LIN {X 0,Y 149.454,Z 1124.639,A -85,B 0,C 180,E1 26452.481,E2 26452.481} C_VEL
LIN {X 0,Y 187.503,Z 1102.336,A -85,B 0,C 180,E1 26457.86,E2 26457.86} C_VEL
LIN {X 0,Y 200.138,Z 1093.431,A -85,B 0,C 180,E1 26459.166,E2 26459.166} C_VEL
LIN {X 0,Y 164.642,Z 1117.097,A -85,B 0,C 180,E1 26463.123,E2 26463.123} C_VEL
LIN {X 0,Y 149.261,Z 1125.368,A -85,B 0,C 180,E1 26463.863,E2 26463.863} C_VEL
LIN {X 0,Y 133.576,Z 1132.787,A -85,B 0,C 180,E1 26464.835,E2 26464.835} C_VEL
LIN {X 0,Y 93.97,Z 1148.455,A -85,B 0,C 180,E1 26475.529,E2 26475.529} C_VEL
LIN {X 0,Y 59.436,Z 1158.376,A -85,B 0,C 180,E1 26500.391,E2 26500.391} C_VEL
LIN {X 0,Y 47.074,Z 1161.431,A -85,B 0,C 180,E1 26534.085,E2 26534.085} C_VEL
LIN {X 0,Y 46.801,Z 1161.776,A -85,B 0,C 180,E1 26550.002,E2 26550.002} C_VEL
LIN {X 0,Y 51.769,Z 1160.244,A -85,B 0,C 180,E1 26585.663,E2 26585.663} C_VEL
LIN {X 0,Y 74.671,Z 1154.337,A -85,B 0,C 180,E1 26614.388,E2 26614.388} C_VEL
LIN {X 0,Y 111.047,Z 1142.33,A -85,B 0,C 180,E1 26630.135,E2 26630.135} C_VEL
LIN {X 0,Y 148.291,Z 1125.731,A -85,B 0,C 180,E1 26637.593,E2 26637.593} C_VEL
LIN {X 0,Y 174.697,Z 1110.81,A -85,B 0,C 180,E1 26640.902,E2 26640.902} C_VEL
LIN {X 0,Y 136.275,Z 1130.859,A -85,B 0,C 180,E1 26646.357,E2 26646.357} C_VEL
LIN {X 0,Y 98.213,Z 1145.413,A -85,B 0,C 180,E1 26656.197,E2 26656.197} C_VEL
LIN {X 0,Y 70.679,Z 1153.183,A -85,B 0,C 180,E1 26671.347,E2 26671.347} C_VEL
LIN {X 0,Y 52.791,Z 1157.045,A -85,B 0,C 180,E1 26695.129,E2 26695.129} C_VEL
LIN {X 0,Y 47.067,Z 1158.256,A -85,B 0,C 180,E1 26729.998,E2 26729.998} C_VEL
LIN {X 0,Y 52.803,Z 1157.02,A -85,B 0,C 180,E1 26764.857,E2 26764.857} C_VEL
LIN {X 0,Y 76.325,Z 1151.652,A -85,B 0,C 180,E1 26792.831,E2 26792.831} C_VEL
LIN {X 0,Y 111.785,Z 1140.677,A -85,B 0,C 180,E1 26808.046,E2 26808.046} C_VEL
LIN {X 0,Y 147.591,Z 1125.471,A -85,B 0,C 180,E1 26815.437,E2 26815.437} C_VEL
LIN {X 0,Y 175.1,Z 1110.402,A -85,B 0,C 180,E1 26819.069,E2 26819.069} C_VEL
LIN {X 0,Y 136.204,Z 1131.534,A -85,B 0,C 180,E1 26824.361,E2 26824.361} C_VEL
LIN {X 0,Y 133.576,Z 1132.787,A -85,B 0,C 180,E1 26824.835,E2 26824.835} C_VEL
LIN {X 0,Y 117.561,Z 1139.427,A -85,B 0,C 180,E1 26826.086,E2 26826.086} C_VEL
LIN {X 0,Y 101.248,Z 1145.06,A -85,B 0,C 180,E1 26827.775,E2 26827.775} C_VEL
LIN {X 0,Y 65.752,Z 1155.495,A -85,B 0,C 180,E1 26843.366,E2 26843.366} C_VEL
LIN {X 0,Y 45.444,Z 1159.922,A -85,B 0,C 180,E1 26868.387,E2 26868.387} C_VEL
LIN {X 0,Y 38.865,Z 1161.478,A -85,B 0,C 180,E1 26910.002,E2 26910.002} C_VEL
LIN {X 0,Y 45.424,Z 1159.939,A -85,B 0,C 180,E1 26951.64,E2 26951.64} C_VEL
LIN {X 0,Y 71.119,Z 1154.125,A -85,B 0,C 180,E1 26980.136,E2 26980.136} C_VEL
LIN {X 0,Y 109.867,Z 1142.045,A -85,B 0,C 180,E1 26994.372,E2 26994.372} C_VEL
LIN {X 0,Y 145.474,Z 1126.776,A -85,B 0,C 180,E1 27000.453,E2 27000.453} C_VEL
LIN {X 0,Y 146.961,Z 1126.007,A -85,B 0,C 180,E1 27001.331,E2 27001.331} C_VEL
LIN {X 0,Y 106.829,Z 1142.355,A -85,B 0,C 180,E1 27008.582,E2 27008.582} C_VEL
LIN {X 0,Y 66.813,Z 1153.487,A -85,B 0,C 180,E1 27025.385,E2 27025.385} C_VEL
LIN {X 0,Y 46.426,Z 1157.346,A -85,B 0,C 180,E1 27049.45,E2 27049.45} C_VEL
LIN {X 0,Y 39.139,Z 1158.553,A -85,B 0,C 180,E1 27089.998,E2 27089.998} C_VEL
LIN {X 0,Y 46.437,Z 1157.322,A -85,B 0,C 180,E1 27130.533,E2 27130.533} C_VEL
LIN {X 0,Y 72.977,Z 1151.957,A -85,B 0,C 180,E1 27158.511,E2 27158.511} C_VEL
LIN {X 0,Y 110.045,Z 1141.106,A -85,B 0,C 180,E1 27172.119,E2 27172.119} C_VEL
LIN {X 0,Y 147.33,Z 1125.697,A -85,B 0,C 180,E1 27178.641,E2 27178.641} C_VEL
LIN {X 0,Y 142.094,Z 1128.261,A -85,B 0,C 180,E1 27180.001,E2 27180.001} C_VEL
LIN {X 0,Y 101.248,Z 1145.06,A -85,B 0,C 180,E1 27187.775,E2 27187.775} C_VEL
LIN {X 0,Y 84.799,Z 1149.904,A -85,B 0,C 180,E1 27190.128,E2 27190.128} C_VEL
LIN {X 0,Y 68.317,Z 1153.871,A -85,B 0,C 180,E1 27193.566,E2 27193.566} C_VEL
LIN {X 0,Y 39.737,Z 1159.617,A -85,B 0,C 180,E1 27220.582,E2 27220.582} C_VEL
LIN {X 0,Y 30.903,Z 1161.18,A -85,B 0,C 180,E1 27270.003,E2 27270.003} C_VEL
LIN {X 0,Y 39.725,Z 1159.635,A -85,B 0,C 180,E1 27319.444,E2 27319.444} C_VEL
LIN {X 0,Y 71.277,Z 1153.213,A -85,B 0,C 180,E1 27347.777,E2 27347.777} C_VEL
LIN {X 0,Y 111.297,Z 1141.025,A -85,B 0,C 180,E1 27359.052,E2 27359.052} C_VEL
LIN {X 0,Y 120.729,Z 1137.474,A -85,B 0,C 180,E1 27360.603,E2 27360.603} C_VEL
LIN {X 0,Y 120.765,Z 1137.402,A -85,B 0,C 180,E1 27361.518,E2 27361.518} C_VEL
LIN {X 0,Y 77.228,Z 1150.824,A -85,B 0,C 180,E1 27372.312,E2 27372.312} C_VEL
LIN {X 0,Y 51.329,Z 1156.057,A -85,B 0,C 180,E1 27388.117,E2 27388.117} C_VEL
LIN {X 0,Y 31.981,Z 1158.66,A -85,B 0,C 180,E1 27430.668,E2 27430.668} C_VEL
LIN {X 0,Y 31.207,Z 1158.851,A -85,B 0,C 180,E1 27449.997,E2 27449.997} C_VEL
LIN {X 0,Y 40.676,Z 1157.623,A -85,B 0,C 180,E1 27497.896,E2 27497.896} C_VEL
LIN {X 0,Y 70.405,Z 1152.263,A -85,B 0,C 180,E1 27524.684,E2 27524.684} C_VEL
LIN {X 0,Y 109.227,Z 1141.412,A -85,B 0,C 180,E1 27536.354,E2 27536.354} C_VEL
LIN {X 0,Y 124.143,Z 1135.961,A -85,B 0,C 180,E1 27538.932,E2 27538.932} C_VEL
LIN {X 0,Y 83.719,Z 1149.879,A -85,B 0,C 180,E1 27547.544,E2 27547.544} C_VEL
LIN {X 0,Y 68.317,Z 1153.871,A -85,B 0,C 180,E1 27553.566,E2 27553.566} C_VEL
LIN {X 0,Y 60.405,Z 1155.568,A -85,B 0,C 180,E1 27556.58,E2 27556.58} C_VEL
LIN {X 0,Y 37.809,Z 1158.877,A -85,B 0,C 180,E1 27566.602,E2 27566.602} C_VEL
LIN {X 0,Y 36.108,Z 1159.131,A -85,B 0,C 180,E1 27568.738,E2 27568.738} C_VEL
LIN {X 0,Y 22.942,Z 1160.881,A -85,B 0,C 180,E1 27630.004,E2 27630.004} C_VEL
LIN {X 0,Y 34.99,Z 1159.331,A -85,B 0,C 180,E1 27689.608,E2 27689.608} C_VEL
LIN {X 0,Y 69.996,Z 1152.904,A -85,B 0,C 180,E1 27714.392,E2 27714.392} C_VEL
LIN {X 0,Y 97.488,Z 1145.407,A -85,B 0,C 180,E1 27721.182,E2 27721.182} C_VEL
LIN {X 0,Y 61.617,Z 1154.096,A -85,B 0,C 180,E1 27731.584,E2 27731.584} C_VEL
LIN {X 0,Y 35.766,Z 1157.948,A -85,B 0,C 180,E1 27752.45,E2 27752.45} C_VEL
LIN {X 0,Y 23.285,Z 1159.148,A -85,B 0,C 180,E1 27809.996,E2 27809.996} C_VEL
LIN {X 0,Y 35.783,Z 1157.925,A -85,B 0,C 180,E1 27867.5,E2 27867.5} C_VEL
LIN {X 0,Y 68.707,Z 1152.568,A -85,B 0,C 180,E1 27891.233,E2 27891.233} C_VEL
LIN {X 0,Y 97.749,Z 1145.252,A -85,B 0,C 180,E1 27898.776,E2 27898.776} C_VEL
LIN {X 0,Y 61.121,Z 1154.877,A -85,B 0,C 180,E1 27909.055,E2 27909.055} C_VEL
LIN {X 0,Y 36.108,Z 1159.131,A -85,B 0,C 180,E1 27928.738,E2 27928.738} C_VEL
LIN {X 0,Y 25.973,Z 1160.253,A -85,B 0,C 180,E1 27944.173,E2 27944.173} C_VEL
LIN {X 0,Y 14.886,Z 1160.49,A -85,B 0,C 180,E1 28002.988,E2 28002.988} C_VEL
LIN {X 0,Y 31.673,Z 1159.027,A -85,B 0,C 180,E1 28062.349,E2 28062.349} C_VEL
LIN {X 0,Y 65.095,Z 1153.591,A -85,B 0,C 180,E1 28079.999,E2 28079.999} C_VEL
LIN {X 0,Y 69.447,Z 1152.63,A -85,B 0,C 180,E1 28081.486,E2 28081.486} C_VEL
LIN {X 0,Y 32.172,Z 1158.25,A -85,B 0,C 180,E1 28100.261,E2 28100.261} C_VEL
LIN {X 0,Y 15.347,Z 1159.445,A -85,B 0,C 180,E1 28169.994,E2 28169.994} C_VEL
LIN {X 0,Y 32.181,Z 1158.227,A -85,B 0,C 180,E1 28239.682,E2 28239.682} C_VEL
LIN {X 0,Y 69.69,Z 1152.528,A -85,B 0,C 180,E1 28258.477,E2 28258.477} C_VEL
LIN {X 0,Y 31.546,Z 1159.018,A -85,B 0,C 180,E1 28277.815,E2 28277.815} C_VEL
LIN {X 0,Y 14.996,Z 1160.583,A -85,B 0,C 180,E1 28350.006,E2 28350.006} C_VEL
LIN {X 0,Y 14.886,Z 1160.49,A -85,B 0,C 180,E1 28362.988,E2 28362.988} C_VEL
LIN {X 0,Y 18.5,Z 1160.034,A -85,B 0,C 180,E1 28407.464,E2 28407.464} C_VEL
LIN {X 0,Y 35.261,Z 1158.109,A -85,B 0,C 180,E1 28439.737,E2 28439.737} C_VEL
LIN {X 0,Y 30.339,Z 1158.552,A -85,B 0,C 180,E1 28445.842,E2 28445.842} C_VEL
LIN {X 0,Y 7.425,Z 1159.742,A -85,B 0,C 180,E1 28529.988,E2 28529.988} C_VEL
LIN {X 0,Y 30.34,Z 1158.529,A -85,B 0,C 180,E1 28614.098,E2 28614.098} C_VEL
LIN {X 0,Y 35.919,Z 1158.001,A -85,B 0,C 180,E1 28620.002,E2 28620.002} C_VEL
LIN {X 0,Y 15.809,Z 1159.852,A -85,B 0,C 180,E1 28637.368,E2 28637.368} C_VEL
LIN {X 0,Y 7.024,Z 1160.224,A -85,B 0,C 180,E1 28727.76,E2 28727.76} C_VEL
LIN {X 0,Y 35.261,Z 1158.109,A -85,B 0,C 180,E1 28799.737,E2 28799.737} C_VEL
LIN {X 0,Y 37.427,Z 1160.095,A -85,B 0,C 180,E1 28800.594,E2 28800.594} C_VEL
LIN {X 0,Y 37.427,Z 1180,A -85,B 0,C 180,E1 28800.594,E2 28800.594} C_VEL
LIN {X 0,Y 37.427,Z 1180,A -85,B 0,C 180,E1 28800.594,E2 28800.594}

QRS_NEXT_CUT()
PTP {E1 28976.914,E2 28976.914}
PTP {X 0,Y 607.928,A -85,B 0,C 180,E1 28976.914,E2 28976.914,E3 0,E4 0,E5 0,E6 0}
QRS_SPEED_INIT()
LIN {X 0,Y 607.928,Z 1180,A -85,B 0,C 180,E1 28976.914,E2 28976.914,E3 0,E4 0,E5 0,E6 0} C_VEL
LIN {X 0,Y 607.928,Z 517.391,A -85,B 0,C 180,E1 28976.914,E2 28976.914} C_VEL
LIN {X 0,Y 607.928,Z 509.317,A -85,B 0,C 180,E1 28976.914,E2 28976.914} C_VEL
LIN {X 0,Y 607.913,Z 507.317,A -85,B 0,C 180,E1 28976.725,E2 28976.725} C_VEL
LIN {X 0,Y 607.889,Z 507.324,A -85,B 0,C 180,E1 28973.483,E2 28973.483} C_VEL
LIN {X 0,Y 607.912,Z 507.317,A -85,B 0,C 180,E1 28970.342,E2 28970.342} C_VEL
LIN {X 0,Y 607.881,Z 507.324,A -85,B 0,C 180,E1 28967.17,E2 28967.17} C_VEL
LIN {X 0,Y 607.916,Z 507.317,A -85,B 0,C 180,E1 28964.057,E2 28964.057} C_VEL
LIN {X 0,Y 607.875,Z 507.324,A -85,B 0,C 180,E1 28960.893,E2 28960.893} C_VEL
LIN {X 0,Y 607.918,Z 507.318,A -85,B 0,C 180,E1 28957.772,E2 28957.772} C_VEL
LIN {X 0,Y 607.866,Z 507.324,A -85,B 0,C 180,E1 28954.561,E2 28954.561} C_VEL
LIN {X 0,Y 607.905,Z 507.319,A -85,B 0,C 180,E1 28951.511,E2 28951.511} C_VEL
LIN {X 0,Y 607.862,Z 507.325,A -85,B 0,C 180,E1 28948.351,E2 28948.351} C_VEL
LIN {X 0,Y 607.873,Z 507.321,A -85,B 0,C 180,E1 28945.426,E2 28945.426} C_VEL
LIN {X 0,Y 607.859,Z 507.326,A -85,B 0,C 180,E1 28942.144,E2 28942.144} C_VEL
LIN {X 0,Y 607.85,Z 507.324,A -85,B 0,C 180,E1 28939.316,E2 28939.316} C_VEL
LIN {X 0,Y 607.874,Z 507.327,A -85,B 0,C 180,E1 28936.092,E2 28936.092} C_VEL
LIN {X 0,Y 607.831,Z 507.325,A -85,B 0,C 180,E1 28933.311,E2 28933.311} C_VEL
LIN {X 0,Y 607.892,Z 507.326,A -85,B 0,C 180,E1 28930.395,E2 28930.395} C_VEL
LIN {X 0,Y 607.869,Z 507.36,A -85,B 0,C 180,E1 28927.756,E2 28927.756} C_VEL
LIN {X 0,Y 607.828,Z 513.922,A -85,B 0,C 180,E1 28927.314,E2 28927.314} C_VEL
LIN {X 0,Y 607.87,Z 686.597,A -85,B 0,C 180,E1 28924.837,E2 28924.837} C_VEL
LIN {X 0,Y 607.91,Z 860.907,A -85,B 0,C 180,E1 28922.383,E2 28922.383} C_VEL
LIN {X 0,Y 607.916,Z 884.698,A -85,B 0,C 180,E1 28921.868,E2 28921.868} C_VEL
LIN {X 0,Y 607.914,Z 903.608,A -85,B 0,C 180,E1 28921.315,E2 28921.315} C_VEL
LIN {X 0,Y 607.913,Z 925.611,A -85,B 0,C 180,E1 28920.511,E2 28920.511} C_VEL
LIN {X 0,Y 607.917,Z 945.361,A -85,B 0,C 180,E1 28919.62,E2 28919.62} C_VEL
LIN {X 0,Y 607.915,Z 966.084,A -85,B 0,C 180,E1 28918.526,E2 28918.526} C_VEL
LIN {X 0,Y 607.915,Z 985.48,A -85,B 0,C 180,E1 28917.315,E2 28917.315} C_VEL
LIN {X 0,Y 607.909,Z 1005.48,A -85,B 0,C 180,E1 28915.884,E2 28915.884} C_VEL
LIN {X 0,Y 607.907,Z 1023.095,A -85,B 0,C 180,E1 28914.435,E2 28914.435} C_VEL
LIN {X 0,Y 607.904,Z 1041.161,A -85,B 0,C 180,E1 28912.738,E2 28912.738} C_VEL
LIN {X 0,Y 607.91,Z 1057.345,A -85,B 0,C 180,E1 28911.012,E2 28911.012} C_VEL
LIN {X 0,Y 607.918,Z 1072.084,A -85,B 0,C 180,E1 28909.205,E2 28909.205} C_VEL
LIN {X 0,Y 607.916,Z 1086.221,A -85,B 0,C 180,E1 28907.221,E2 28907.221} C_VEL
LIN {X 0,Y 607.896,Z 1097.766,A -85,B 0,C 180,E1 28905.356,E2 28905.356} C_VEL
LIN {X 0,Y 607.887,Z 1108.537,A -85,B 0,C 180,E1 28903.313,E2 28903.313} C_VEL
LIN {X 0,Y 607.912,Z 1117.182,A -85,B 0,C 180,E1 28901.383,E2 28901.383} C_VEL
LIN {X 0,Y 607.892,Z 1124.893,A -85,B 0,C 180,E1 28899.276,E2 28899.276} C_VEL
LIN {X 0,Y 607.89,Z 1130.468,A -85,B 0,C 180,E1 28897.371,E2 28897.371} C_VEL
LIN {X 0,Y 607.911,Z 1135.403,A -85,B 0,C 180,E1 28895.096,E2 28895.096} C_VEL
LIN {X 0,Y 607.881,Z 1138.125,A -85,B 0,C 180,E1 28893.206,E2 28893.206} C_VEL
LIN {X 0,Y 607.901,Z 1139.75,A -85,B 0,C 180,E1 28891.037,E2 28891.037} C_VEL
LIN {X 0,Y 607.886,Z 1139.794,A -85,B 0,C 180,E1 28889.058,E2 28889.058} C_VEL
LIN {X 0,Y 607.883,Z 1138.346,A -85,B 0,C 180,E1 28886.889,E2 28886.889} C_VEL
LIN {X 0,Y 607.905,Z 1135.714,A -85,B 0,C 180,E1 28884.999,E2 28884.999} C_VEL
LIN {X 0,Y 607.88,Z 1131.475,A -85,B 0,C 180,E1 28882.914,E2 28882.914} C_VEL
LIN {X 0,Y 607.914,Z 1125.791,A -85,B 0,C 180,E1 28880.915,E2 28880.915} C_VEL
LIN {X 0,Y 607.898,Z 1118.365,A -85,B 0,C 180,E1 28878.809,E2 28878.809} C_VEL
LIN {X 0,Y 607.89,Z 1109.434,A -85,B 0,C 180,E1 28876.784,E2 28876.784} C_VEL
LIN {X 0,Y 607.913,Z 1099.426,A -85,B 0,C 180,E1 28874.84,E2 28874.84} C_VEL
LIN {X 0,Y 607.914,Z 1087.341,A -85,B 0,C 180,E1 28872.861,E2 28872.861} C_VEL
LIN {X 0,Y 607.914,Z 1074.345,A -85,B 0,C 180,E1 28870.995,E2 28870.995} C_VEL
LIN {X 0,Y 607.907,Z 1059.812,A -85,B 0,C 180,E1 28869.19,E2 28869.19} C_VEL
LIN {X 0,Y 607.902,Z 1042.699,A -85,B 0,C 180,E1 28867.326,E2 28867.326} C_VEL
LIN {X 0,Y 607.905,Z 1025.391,A -85,B 0,C 180,E1 28865.671,E2 28865.671} C_VEL
LIN {X 0,Y 607.908,Z 1007.176,A -85,B 0,C 180,E1 28864.16,E2 28864.16} C_VEL
LIN {X 0,Y 607.914,Z 986.209,A -85,B 0,C 180,E1 28862.643,E2 28862.643} C_VEL
LIN {X 0,Y 607.917,Z 966.952,A -85,B 0,C 180,E1 28861.436,E2 28861.436} C_VEL
LIN {X 0,Y 607.918,Z 946.109,A -85,B 0,C 180,E1 28860.326,E2 28860.326} C_VEL
LIN {X 0,Y 607.914,Z 926.897,A -85,B 0,C 180,E1 28859.454,E2 28859.454} C_VEL
LIN {X 0,Y 607.913,Z 905.218,A -85,B 0,C 180,E1 28858.646,E2 28858.646} C_VEL
LIN {X 0,Y 607.917,Z 886.885,A -85,B 0,C 180,E1 28858.1,E2 28858.1} C_VEL
LIN {X 0,Y 607.912,Z 865.475,A -85,B 0,C 180,E1 28857.604,E2 28857.604} C_VEL
LIN {X 0,Y 607.912,Z 827.721,A -85,B 0,C 180,E1 28857.044,E2 28857.044} C_VEL
LIN {X 0,Y 607.905,Z 618.938,A -85,B 0,C 180,E1 28854.116,E2 28854.116} C_VEL
LIN {X 0,Y 607.834,Z 512.994,A -85,B 0,C 180,E1 28852.56,E2 28852.56} C_VEL
LIN {X 0,Y 607.877,Z 507.33,A -85,B 0,C 180,E1 28852.141,E2 28852.141} C_VEL
LIN {X 0,Y 607.826,Z 507.328,A -85,B 0,C 180,E1 28848.978,E2 28848.978} C_VEL
LIN {X 0,Y 607.837,Z 507.328,A -85,B 0,C 180,E1 28846.231,E2 28846.231} C_VEL
LIN {X 0,Y 607.853,Z 507.326,A -85,B 0,C 180,E1 28842.921,E2 28842.921} C_VEL
LIN {X 0,Y 607.834,Z 507.326,A -85,B 0,C 180,E1 28840.248,E2 28840.248} C_VEL
LIN {X 0,Y 607.91,Z 507.328,A -85,B 0,C 180,E1 28837.245,E2 28837.245} C_VEL
LIN {X 0,Y 607.844,Z 507.324,A -85,B 0,C 180,E1 28834.12,E2 28834.12} C_VEL
LIN {X 0,Y 607.896,Z 507.327,A -85,B 0,C 180,E1 28831.206,E2 28831.206} C_VEL
LIN {X 0,Y 607.862,Z 507.322,A -85,B 0,C 180,E1 28828.063,E2 28828.063} C_VEL
LIN {X 0,Y 607.882,Z 507.326,A -85,B 0,C 180,E1 28825.111,E2 28825.111} C_VEL
LIN {X 0,Y 607.875,Z 507.321,A -85,B 0,C 180,E1 28821.823,E2 28821.823} C_VEL
LIN {X 0,Y 607.891,Z 507.326,A -85,B 0,C 180,E1 28818.807,E2 28818.807} C_VEL
LIN {X 0,Y 607.885,Z 507.319,A -85,B 0,C 180,E1 28815.552,E2 28815.552} C_VEL
LIN {X 0,Y 607.906,Z 507.327,A -85,B 0,C 180,E1 28812.443,E2 28812.443} C_VEL
LIN {X 0,Y 607.887,Z 507.319,A -85,B 0,C 180,E1 28809.181,E2 28809.181} C_VEL
LIN {X 0,Y 607.917,Z 507.326,A -85,B 0,C 180,E1 28806.043,E2 28806.043} C_VEL
LIN {X 0,Y 607.89,Z 507.319,A -85,B 0,C 180,E1 28802.829,E2 28802.829} C_VEL
LIN {X 0,Y 607.909,Z 507.326,A -85,B 0,C 180,E1 28799.718,E2 28799.718} C_VEL
LIN {X 0,Y 607.896,Z 507.318,A -85,B 0,C 180,E1 28796.511,E2 28796.511} C_VEL
LIN {X 0,Y 607.903,Z 507.325,A -85,B 0,C 180,E1 28793.389,E2 28793.389} C_VEL
LIN {X 0,Y 607.899,Z 507.319,A -85,B 0,C 180,E1 28790.151,E2 28790.151} C_VEL
LIN {X 0,Y 607.893,Z 507.323,A -85,B 0,C 180,E1 28786.978,E2 28786.978} C_VEL
LIN {X 0,Y 607.904,Z 507.319,A -85,B 0,C 180,E1 28783.852,E2 28783.852} C_VEL
LIN {X 0,Y 607.887,Z 507.323,A -85,B 0,C 180,E1 28780.695,E2 28780.695} C_VEL
LIN {X 0,Y 607.908,Z 507.319,A -85,B 0,C 180,E1 28777.569,E2 28777.569} C_VEL
LIN {X 0,Y 607.879,Z 507.323,A -85,B 0,C 180,E1 28774.368,E2 28774.368} C_VEL
LIN {X 0,Y 607.912,Z 507.319,A -85,B 0,C 180,E1 28771.241,E2 28771.241} C_VEL
LIN {X 0,Y 607.871,Z 507.323,A -85,B 0,C 180,E1 28768.076,E2 28768.076} C_VEL
LIN {X 0,Y 607.916,Z 507.319,A -85,B 0,C 180,E1 28764.97,E2 28764.97} C_VEL
LIN {X 0,Y 607.864,Z 507.323,A -85,B 0,C 180,E1 28761.796,E2 28761.796} C_VEL
LIN {X 0,Y 607.911,Z 507.32,A -85,B 0,C 180,E1 28758.733,E2 28758.733} C_VEL
LIN {X 0,Y 607.857,Z 507.325,A -85,B 0,C 180,E1 28755.552,E2 28755.552} C_VEL
LIN {X 0,Y 607.879,Z 507.323,A -85,B 0,C 180,E1 28752.662,E2 28752.662} C_VEL
LIN {X 0,Y 607.891,Z 507.532,A -85,B 0,C 180,E1 28749.751,E2 28749.751} C_VEL
LIN {X 0,Y 607.863,Z 542.978,A -85,B 0,C 180,E1 28747.37,E2 28747.37} C_VEL
LIN {X 0,Y 607.877,Z 722.13,A -85,B 0,C 180,E1 28744.803,E2 28744.803} C_VEL
LIN {X 0,Y 607.912,Z 891.131,A -85,B 0,C 180,E1 28742.424,E2 28742.424} C_VEL
LIN {X 0,Y 607.916,Z 913.981,A -85,B 0,C 180,E1 28741.932,E2 28741.932} C_VEL
LIN {X 0,Y 607.915,Z 932.562,A -85,B 0,C 180,E1 28741.394,E2 28741.394} C_VEL
LIN {X 0,Y 607.912,Z 953.928,A -85,B 0,C 180,E1 28740.628,E2 28740.628} C_VEL
LIN {X 0,Y 607.919,Z 974.107,A -85,B 0,C 180,E1 28739.726,E2 28739.726} C_VEL
LIN {X 0,Y 607.916,Z 994.762,A -85,B 0,C 180,E1 28738.649,E2 28738.649} C_VEL
LIN {X 0,Y 607.917,Z 1014.564,A -85,B 0,C 180,E1 28737.421,E2 28737.421} C_VEL
LIN {X 0,Y 607.912,Z 1033.959,A -85,B 0,C 180,E1 28736.049,E2 28736.049} C_VEL
LIN {X 0,Y 607.91,Z 1052.18,A -85,B 0,C 180,E1 28734.558,E2 28734.558} C_VEL
LIN {X 0,Y 607.904,Z 1070.598,A -85,B 0,C 180,E1 28732.84,E2 28732.84} C_VEL
LIN {X 0,Y 607.916,Z 1086.876,A -85,B 0,C 180,E1 28731.112,E2 28731.112} C_VEL
LIN {X 0,Y 607.917,Z 1102.056,A -85,B 0,C 180,E1 28729.254,E2 28729.254} C_VEL
LIN {X 0,Y 607.916,Z 1116.517,A -85,B 0,C 180,E1 28727.221,E2 28727.221} C_VEL
LIN {X 0,Y 607.9,Z 1128.035,A -85,B 0,C 180,E1 28725.355,E2 28725.355} C_VEL
LIN {X 0,Y 607.886,Z 1138.755,A -85,B 0,C 180,E1 28723.313,E2 28723.313} C_VEL
LIN {X 0,Y 607.909,Z 1147.375,A -85,B 0,C 180,E1 28721.383,E2 28721.383} C_VEL
LIN {X 0,Y 607.896,Z 1155.038,A -85,B 0,C 180,E1 28719.276,E2 28719.276} C_VEL
LIN {X 0,Y 607.888,Z 1160.59,A -85,B 0,C 180,E1 28717.371,E2 28717.371} C_VEL
LIN {X 0,Y 607.91,Z 1165.479,A -85,B 0,C 180,E1 28715.095,E2 28715.095} C_VEL
LIN {X 0,Y 607.881,Z 1168.179,A -85,B 0,C 180,E1 28713.206,E2 28713.206} C_VEL
LIN {X 0,Y 607.897,Z 1169.761,A -85,B 0,C 180,E1 28711.036,E2 28711.036} C_VEL
LIN {X 0,Y 607.886,Z 1169.805,A -85,B 0,C 180,E1 28709.152,E2 28709.152} C_VEL
LIN {X 0,Y 607.884,Z 1168.404,A -85,B 0,C 180,E1 28706.983,E2 28706.983} C_VEL
LIN {X 0,Y 607.909,Z 1165.638,A -85,B 0,C 180,E1 28704.999,E2 28704.999} C_VEL
LIN {X 0,Y 607.882,Z 1161.099,A -85,B 0,C 180,E1 28702.819,E2 28702.819} C_VEL
LIN {X 0,Y 607.913,Z 1155.646,A -85,B 0,C 180,E1 28700.915,E2 28700.915} C_VEL
LIN {X 0,Y 607.901,Z 1148.186,A -85,B 0,C 180,E1 28698.809,E2 28698.809} C_VEL
LIN {X 0,Y 607.887,Z 1139.217,A -85,B 0,C 180,E1 28696.783,E2 28696.783} C_VEL
LIN {X 0,Y 607.912,Z 1129.179,A -85,B 0,C 180,E1 28694.84,E2 28694.84} C_VEL
LIN {X 0,Y 607.916,Z 1117.035,A -85,B 0,C 180,E1 28692.859,E2 28692.859} C_VEL
LIN {X 0,Y 607.916,Z 1103.213,A -85,B 0,C 180,E1 28690.895,E2 28690.895} C_VEL
LIN {X 0,Y 607.907,Z 1088.576,A -85,B 0,C 180,E1 28689.089,E2 28689.089} C_VEL
LIN {X 0,Y 607.901,Z 1072.244,A -85,B 0,C 180,E1 28687.326,E2 28687.326} C_VEL
LIN {X 0,Y 607.905,Z 1054.853,A -85,B 0,C 180,E1 28685.67,E2 28685.67} C_VEL
LIN {X 0,Y 607.908,Z 1036.601,A -85,B 0,C 180,E1 28684.16,E2 28684.16} C_VEL
LIN {X 0,Y 607.913,Z 1016.161,A -85,B 0,C 180,E1 28682.685,E2 28682.685} C_VEL
LIN {X 0,Y 607.915,Z 996.826,A -85,B 0,C 180,E1 28681.474,E2 28681.474} C_VEL
LIN {X 0,Y 607.918,Z 976.29,A -85,B 0,C 180,E1 28680.38,E2 28680.38} C_VEL
LIN {X 0,Y 607.914,Z 957.45,A -85,B 0,C 180,E1 28679.523,E2 28679.523} C_VEL
LIN {X 0,Y 607.913,Z 935.014,A -85,B 0,C 180,E1 28678.685,E2 28678.685} C_VEL
LIN {X 0,Y 607.915,Z 916.38,A -85,B 0,C 180,E1 28678.132,E2 28678.132} C_VEL
LIN {X 0,Y 607.912,Z 894.525,A -85,B 0,C 180,E1 28677.631,E2 28677.631} C_VEL
LIN {X 0,Y 607.912,Z 851.351,A -85,B 0,C 180,E1 28677.001,E2 28677.001} C_VEL
LIN {X 0,Y 607.907,Z 642.697,A -85,B 0,C 180,E1 28674.072,E2 28674.072} C_VEL
LIN {X 0,Y 607.865,Z 542.542,A -85,B 0,C 180,E1 28672.605,E2 28672.605} C_VEL
LIN {X 0,Y 607.894,Z 507.329,A -85,B 0,C 180,E1 28670.221,E2 28670.221} C_VEL
LIN {X 0,Y 607.856,Z 507.324,A -85,B 0,C 180,E1 28667.052,E2 28667.052} C_VEL
LIN {X 0,Y 607.874,Z 507.326,A -85,B 0,C 180,E1 28664.179,E2 28664.179} C_VEL
LIN {X 0,Y 607.874,Z 507.321,A -85,B 0,C 180,E1 28660.893,E2 28660.893} C_VEL
LIN {X 0,Y 607.884,Z 507.326,A -85,B 0,C 180,E1 28657.859,E2 28657.859} C_VEL
LIN {X 0,Y 607.88,Z 507.319,A -85,B 0,C 180,E1 28654.573,E2 28654.573} C_VEL
LIN {X 0,Y 607.894,Z 507.326,A -85,B 0,C 180,E1 28651.536,E2 28651.536} C_VEL
LIN {X 0,Y 607.887,Z 507.319,A -85,B 0,C 180,E1 28648.275,E2 28648.275} C_VEL
LIN {X 0,Y 607.912,Z 507.328,A -85,B 0,C 180,E1 28645.109,E2 28645.109} C_VEL
LIN {X 0,Y 607.885,Z 507.319,A -85,B 0,C 180,E1 28641.822,E2 28641.822} C_VEL
LIN {X 0,Y 607.91,Z 507.324,A -85,B 0,C 180,E1 28638.669,E2 28638.669} C_VEL
LIN {X 0,Y 607.889,Z 507.319,A -85,B 0,C 180,E1 28635.45,E2 28635.45} C_VEL
LIN {X 0,Y 607.903,Z 507.323,A -85,B 0,C 180,E1 28632.312,E2 28632.312} C_VEL
LIN {X 0,Y 607.896,Z 507.318,A -85,B 0,C 180,E1 28629.18,E2 28629.18} C_VEL
LIN {X 0,Y 607.899,Z 507.324,A -85,B 0,C 180,E1 28626.042,E2 28626.042} C_VEL
LIN {X 0,Y 607.901,Z 507.318,A -85,B 0,C 180,E1 28622.922,E2 28622.922} C_VEL
LIN {X 0,Y 607.896,Z 507.324,A -85,B 0,C 180,E1 28619.811,E2 28619.811} C_VEL
LIN {X 0,Y 607.913,Z 507.317,A -85,B 0,C 180,E1 28616.725,E2 28616.725} C_VEL
LIN {X 0,Y 606.9,Z 507.453,A -85,B 0,C 180,E1 28615.999,E2 28615.999} C_VEL
LIN {X 0,Y 600.49,Z 508.252,A -85,B 0,C 180,E1 28613.963,E2 28613.963} C_VEL
LIN {X 0,Y 599.948,Z 508.313,A -85,B 0,C 180,E1 28613.433,E2 28613.433} C_VEL
LIN {X 0,Y 599.972,Z 508.306,A -85,B 0,C 180,E1 28610.31,E2 28610.31} C_VEL
LIN {X 0,Y 599.94,Z 508.312,A -85,B 0,C 180,E1 28607.095,E2 28607.095} C_VEL
LIN {X 0,Y 599.973,Z 508.308,A -85,B 0,C 180,E1 28603.94,E2 28603.94} C_VEL
LIN {X 0,Y 599.934,Z 508.313,A -85,B 0,C 180,E1 28600.833,E2 28600.833} C_VEL
LIN {X 0,Y 599.979,Z 508.307,A -85,B 0,C 180,E1 28597.772,E2 28597.772} C_VEL
LIN {X 0,Y 599.926,Z 508.313,A -85,B 0,C 180,E1 28594.533,E2 28594.533} C_VEL
LIN {X 0,Y 599.977,Z 508.308,A -85,B 0,C 180,E1 28591.426,E2 28591.426} C_VEL
LIN {X 0,Y 599.918,Z 508.314,A -85,B 0,C 180,E1 28588.212,E2 28588.212} C_VEL
LIN {X 0,Y 599.953,Z 508.309,A -85,B 0,C 180,E1 28585.248,E2 28585.248} C_VEL
LIN {X 0,Y 599.913,Z 508.314,A -85,B 0,C 180,E1 28582.031,E2 28582.031} C_VEL
LIN {X 0,Y 599.921,Z 508.313,A -85,B 0,C 180,E1 28579.171,E2 28579.171} C_VEL
LIN {X 0,Y 599.911,Z 508.316,A -85,B 0,C 180,E1 28575.839,E2 28575.839} C_VEL
LIN {X 0,Y 599.897,Z 508.312,A -85,B 0,C 180,E1 28573.107,E2 28573.107} C_VEL
LIN {X 0,Y 599.946,Z 508.319,A -85,B 0,C 180,E1 28569.948,E2 28569.948} C_VEL
LIN {X 0,Y 599.984,Z 508.535,A -85,B 0,C 180,E1 28568.256,E2 28568.256} C_VEL
LIN {X 0,Y 601.035,Z 511.879,A -85,B 0,C 180,E1 28567.93,E2 28567.93} C_VEL
LIN {X 0,Y 601.19,Z 514.196,A -85,B 0,C 180,E1 28567.794,E2 28567.794} C_VEL
LIN {X 0,Y 601.452,Z 518.798,A -85,B 0,C 180,E1 28567.707,E2 28567.707} C_VEL
LIN {X 0,Y 601.3,Z 691.878,A -85,B 0,C 180,E1 28565.198,E2 28565.198} C_VEL
LIN {X 0,Y 601.144,Z 861.272,A -85,B 0,C 180,E1 28562.788,E2 28562.788} C_VEL
LIN {X 0,Y 601.069,Z 884.986,A -85,B 0,C 180,E1 28562.268,E2 28562.268} C_VEL
LIN {X 0,Y 600.998,Z 904.602,A -85,B 0,C 180,E1 28561.686,E2 28561.686} C_VEL
LIN {X 0,Y 600.875,Z 927.356,A -85,B 0,C 180,E1 28560.832,E2 28560.832} C_VEL
LIN {X 0,Y 600.792,Z 946.497,A -85,B 0,C 180,E1 28559.952,E2 28559.952} C_VEL
LIN {X 0,Y 600.649,Z 968.506,A -85,B 0,C 180,E1 28558.756,E2 28558.756} C_VEL
LIN {X 0,Y 600.551,Z 987.9,A -85,B 0,C 180,E1 28557.517,E2 28557.517} C_VEL
LIN {X 0,Y 600.413,Z 1008.027,A -85,B 0,C 180,E1 28556.028,E2 28556.028} C_VEL
LIN {X 0,Y 600.307,Z 1026.656,A -85,B 0,C 180,E1 28554.45,E2 28554.45} C_VEL
LIN {X 0,Y 600.212,Z 1043.702,A -85,B 0,C 180,E1 28552.788,E2 28552.788} C_VEL
LIN {X 0,Y 600.124,Z 1059.906,A -85,B 0,C 180,E1 28550.991,E2 28550.991} C_VEL
LIN {X 0,Y 600.078,Z 1074.623,A -85,B 0,C 180,E1 28549.136,E2 28549.136} C_VEL
LIN {X 0,Y 600.02,Z 1088.156,A -85,B 0,C 180,E1 28547.155,E2 28547.155} C_VEL
LIN {X 0,Y 599.978,Z 1100.511,A -85,B 0,C 180,E1 28545.069,E2 28545.069} C_VEL
LIN {X 0,Y 599.926,Z 1109.933,A -85,B 0,C 180,E1 28543.199,E2 28543.199} C_VEL
LIN {X 0,Y 599.918,Z 1119.102,A -85,B 0,C 180,E1 28541.05,E2 28541.05} C_VEL
LIN {X 0,Y 599.923,Z 1126.115,A -85,B 0,C 180,E1 28539.014,E2 28539.014} C_VEL
LIN {X 0,Y 599.89,Z 1132.123,A -85,B 0,C 180,E1 28536.796,E2 28536.796} C_VEL
LIN {X 0,Y 599.903,Z 1136.041,A -85,B 0,C 180,E1 28534.781,E2 28534.781} C_VEL
LIN {X 0,Y 599.911,Z 1138.821,A -85,B 0,C 180,E1 28532.579,E2 28532.579} C_VEL
LIN {X 0,Y 599.885,Z 1139.862,A -85,B 0,C 180,E1 28530.573,E2 28530.573} C_VEL
LIN {X 0,Y 599.908,Z 1139.623,A -85,B 0,C 180,E1 28528.472,E2 28528.472} C_VEL
LIN {X 0,Y 599.894,Z 1137.781,A -85,B 0,C 180,E1 28526.369,E2 28526.369} C_VEL
LIN {X 0,Y 599.891,Z 1134.587,A -85,B 0,C 180,E1 28524.261,E2 28524.261} C_VEL
LIN {X 0,Y 599.916,Z 1129.689,A -85,B 0,C 180,E1 28522.145,E2 28522.145} C_VEL
LIN {X 0,Y 599.902,Z 1123.343,A -85,B 0,C 180,E1 28520.018,E2 28520.018} C_VEL
LIN {X 0,Y 599.917,Z 1115.52,A -85,B 0,C 180,E1 28517.975,E2 28517.975} C_VEL
LIN {X 0,Y 599.965,Z 1106.148,A -85,B 0,C 180,E1 28515.911,E2 28515.911} C_VEL
LIN {X 0,Y 599.974,Z 1095.397,A -85,B 0,C 180,E1 28513.94,E2 28513.94} C_VEL
LIN {X 0,Y 600.022,Z 1082.895,A -85,B 0,C 180,E1 28511.944,E2 28511.944} C_VEL
LIN {X 0,Y 600.076,Z 1069.672,A -85,B 0,C 180,E1 28510.129,E2 28510.129} C_VEL
LIN {X 0,Y 600.159,Z 1053.603,A -85,B 0,C 180,E1 28508.191,E2 28508.191} C_VEL
LIN {X 0,Y 600.263,Z 1036.98,A -85,B 0,C 180,E1 28506.436,E2 28506.436} C_VEL
LIN {X 0,Y 600.349,Z 1019.31,A -85,B 0,C 180,E1 28504.816,E2 28504.816} C_VEL
LIN {X 0,Y 600.476,Z 999.507,A -85,B 0,C 180,E1 28503.225,E2 28503.225} C_VEL
LIN {X 0,Y 600.577,Z 980.42,A -85,B 0,C 180,E1 28501.891,E2 28501.891} C_VEL
LIN {X 0,Y 600.716,Z 959.629,A -85,B 0,C 180,E1 28500.648,E2 28500.648} C_VEL
LIN {X 0,Y 600.811,Z 939.378,A -85,B 0,C 180,E1 28499.608,E2 28499.608} C_VEL
LIN {X 0,Y 600.94,Z 917.845,A -85,B 0,C 180,E1 28498.699,E2 28498.699} C_VEL
LIN {X 0,Y 601.016,Z 898.164,A -85,B 0,C 180,E1 28498.016,E2 28498.016} C_VEL
LIN {X 0,Y 601.11,Z 875.009,A -85,B 0,C 180,E1 28497.4,E2 28497.4} C_VEL
LIN {X 0,Y 601.155,Z 855.819,A -85,B 0,C 180,E1 28497.033,E2 28497.033} C_VEL
LIN {X 0,Y 601.359,Z 641.166,A -85,B 0,C 180,E1 28493.986,E2 28493.986} C_VEL
LIN {X 0,Y 601.268,Z 514.517,A -85,B 0,C 180,E1 28492.126,E2 28492.126} C_VEL
LIN {X 0,Y 601.031,Z 512.812,A -85,B 0,C 180,E1 28492.049,E2 28492.049} C_VEL
LIN {X 0,Y 600.875,Z 511.129,A -85,B 0,C 180,E1 28491.913,E2 28491.913} C_VEL
LIN {X 0,Y 599.944,Z 508.319,A -85,B 0,C 180,E1 28491.625,E2 28491.625} C_VEL
LIN {X 0,Y 599.881,Z 508.318,A -85,B 0,C 180,E1 28488.697,E2 28488.697} C_VEL
LIN {X 0,Y 599.975,Z 508.317,A -85,B 0,C 180,E1 28485.579,E2 28485.579} C_VEL
LIN {X 0,Y 599.894,Z 508.315,A -85,B 0,C 180,E1 28482.549,E2 28482.549} C_VEL
LIN {X 0,Y 599.935,Z 508.316,A -85,B 0,C 180,E1 28479.666,E2 28479.666} C_VEL
LIN {X 0,Y 599.908,Z 508.314,A -85,B 0,C 180,E1 28476.394,E2 28476.394} C_VEL
LIN {X 0,Y 599.925,Z 508.313,A -85,B 0,C 180,E1 28473.559,E2 28473.559} C_VEL
LIN {X 0,Y 599.925,Z 508.31,A -85,B 0,C 180,E1 28470.22,E2 28470.22} C_VEL
LIN {X 0,Y 599.934,Z 508.314,A -85,B 0,C 180,E1 28467.279,E2 28467.279} C_VEL
LIN {X 0,Y 599.939,Z 508.307,A -85,B 0,C 180,E1 28463.995,E2 28463.995} C_VEL
LIN {X 0,Y 599.941,Z 508.314,A -85,B 0,C 180,E1 28460.997,E2 28460.997} C_VEL
LIN {X 0,Y 599.943,Z 508.306,A -85,B 0,C 180,E1 28457.657,E2 28457.657} C_VEL
LIN {X 0,Y 599.972,Z 508.315,A -85,B 0,C 180,E1 28454.476,E2 28454.476} C_VEL
LIN {X 0,Y 599.944,Z 508.308,A -85,B 0,C 180,E1 28451.244,E2 28451.244} C_VEL
LIN {X 0,Y 599.975,Z 508.314,A -85,B 0,C 180,E1 28448.047,E2 28448.047} C_VEL
LIN {X 0,Y 599.948,Z 508.308,A -85,B 0,C 180,E1 28444.876,E2 28444.876} C_VEL
LIN {X 0,Y 599.969,Z 508.313,A -85,B 0,C 180,E1 28441.719,E2 28441.719} C_VEL
LIN {X 0,Y 599.954,Z 508.308,A -85,B 0,C 180,E1 28438.568,E2 28438.568} C_VEL
LIN {X 0,Y 599.963,Z 508.313,A -85,B 0,C 180,E1 28435.412,E2 28435.412} C_VEL
LIN {X 0,Y 599.959,Z 508.308,A -85,B 0,C 180,E1 28432.242,E2 28432.242} C_VEL
LIN {X 0,Y 599.955,Z 508.309,A -85,B 0,C 180,E1 28429.048,E2 28429.048} C_VEL
LIN {X 0,Y 599.963,Z 508.308,A -85,B 0,C 180,E1 28425.913,E2 28425.913} C_VEL
LIN {X 0,Y 599.947,Z 508.309,A -85,B 0,C 180,E1 28422.737,E2 28422.737} C_VEL
LIN {X 0,Y 599.968,Z 508.308,A -85,B 0,C 180,E1 28419.617,E2 28419.617} C_VEL
LIN {X 0,Y 599.944,Z 508.31,A -85,B 0,C 180,E1 28416.528,E2 28416.528} C_VEL
LIN {X 0,Y 599.973,Z 508.308,A -85,B 0,C 180,E1 28413.366,E2 28413.366} C_VEL
LIN {X 0,Y 599.937,Z 508.312,A -85,B 0,C 180,E1 28410.222,E2 28410.222} C_VEL
LIN {X 0,Y 599.977,Z 508.308,A -85,B 0,C 180,E1 28407.093,E2 28407.093} C_VEL
LIN {X 0,Y 599.929,Z 508.313,A -85,B 0,C 180,E1 28403.932,E2 28403.932} C_VEL
LIN {X 0,Y 599.975,Z 508.307,A -85,B 0,C 180,E1 28400.798,E2 28400.798} C_VEL
LIN {X 0,Y 599.919,Z 508.313,A -85,B 0,C 180,E1 28397.589,E2 28397.589} C_VEL
LIN {X 0,Y 599.975,Z 508.31,A -85,B 0,C 180,E1 28394.5,E2 28394.5} C_VEL
LIN {X 0,Y 599.91,Z 508.317,A -85,B 0,C 180,E1 28391.3,E2 28391.3} C_VEL
LIN {X 0,Y 599.973,Z 508.38,A -85,B 0,C 180,E1 28390.323,E2 28390.323} C_VEL
LIN {X 0,Y 601.235,Z 512.489,A -85,B 0,C 180,E1 28389.935,E2 28389.935} C_VEL
LIN {X 0,Y 601.225,Z 543.474,A -85,B 0,C 180,E1 28387.847,E2 28387.847} C_VEL
LIN {X 0,Y 601.487,Z 548.323,A -85,B 0,C 180,E1 28387.756,E2 28387.756} C_VEL
LIN {X 0,Y 601.301,Z 727.728,A -85,B 0,C 180,E1 28385.16,E2 28385.16} C_VEL
LIN {X 0,Y 601.147,Z 891.238,A -85,B 0,C 180,E1 28382.833,E2 28382.833} C_VEL
LIN {X 0,Y 601.069,Z 914.91,A -85,B 0,C 180,E1 28382.315,E2 28382.315} C_VEL
LIN {X 0,Y 600.998,Z 934.577,A -85,B 0,C 180,E1 28381.731,E2 28381.731} C_VEL
LIN {X 0,Y 600.875,Z 957.254,A -85,B 0,C 180,E1 28380.881,E2 28380.881} C_VEL
LIN {X 0,Y 600.793,Z 976.303,A -85,B 0,C 180,E1 28380.007,E2 28380.007} C_VEL
LIN {X 0,Y 600.656,Z 997.47,A -85,B 0,C 180,E1 28378.864,E2 28378.864} C_VEL
LIN {X 0,Y 600.556,Z 1016.894,A -85,B 0,C 180,E1 28377.63,E2 28377.63} C_VEL
LIN {X 0,Y 600.418,Z 1036.952,A -85,B 0,C 180,E1 28376.159,E2 28376.159} C_VEL
LIN {X 0,Y 600.324,Z 1055.725,A -85,B 0,C 180,E1 28374.581,E2 28374.581} C_VEL
LIN {X 0,Y 600.213,Z 1073.065,A -85,B 0,C 180,E1 28372.898,E2 28372.898} C_VEL
LIN {X 0,Y 600.124,Z 1090.285,A -85,B 0,C 180,E1 28370.99,E2 28370.99} C_VEL
LIN {X 0,Y 600.076,Z 1104.956,A -85,B 0,C 180,E1 28369.137,E2 28369.137} C_VEL
LIN {X 0,Y 600.019,Z 1118.448,A -85,B 0,C 180,E1 28367.154,E2 28367.154} C_VEL
LIN {X 0,Y 599.976,Z 1130.75,A -85,B 0,C 180,E1 28365.068,E2 28365.068} C_VEL
LIN {X 0,Y 599.925,Z 1140.148,A -85,B 0,C 180,E1 28363.199,E2 28363.199} C_VEL
LIN {X 0,Y 599.917,Z 1149.482,A -85,B 0,C 180,E1 28360.991,E2 28360.991} C_VEL
LIN {X 0,Y 599.925,Z 1156.258,A -85,B 0,C 180,E1 28359.013,E2 28359.013} C_VEL
LIN {X 0,Y 599.892,Z 1162.22,A -85,B 0,C 180,E1 28356.796,E2 28356.796} C_VEL
LIN {X 0,Y 599.901,Z 1166.116,A -85,B 0,C 180,E1 28354.78,E2 28354.78} C_VEL
LIN {X 0,Y 599.916,Z 1168.853,A -85,B 0,C 180,E1 28352.579,E2 28352.579} C_VEL
LIN {X 0,Y 599.883,Z 1169.872,A -85,B 0,C 180,E1 28350.573,E2 28350.573} C_VEL
LIN {X 0,Y 599.904,Z 1169.524,A -85,B 0,C 180,E1 28348.376,E2 28348.376} C_VEL
LIN {X 0,Y 599.897,Z 1167.728,A -85,B 0,C 180,E1 28346.368,E2 28346.368} C_VEL
LIN {X 0,Y 599.889,Z 1164.493,A -85,B 0,C 180,E1 28344.26,E2 28344.26} C_VEL
LIN {X 0,Y 599.916,Z 1159.569,A -85,B 0,C 180,E1 28342.145,E2 28342.145} C_VEL
LIN {X 0,Y 599.905,Z 1153.182,A -85,B 0,C 180,E1 28340.018,E2 28340.018} C_VEL
LIN {X 0,Y 599.914,Z 1145.329,A -85,B 0,C 180,E1 28337.975,E2 28337.975} C_VEL
LIN {X 0,Y 599.963,Z 1135.914,A -85,B 0,C 180,E1 28335.91,E2 28335.91} C_VEL
LIN {X 0,Y 599.977,Z 1125.132,A -85,B 0,C 180,E1 28333.94,E2 28333.94} C_VEL
LIN {X 0,Y 600.024,Z 1112.577,A -85,B 0,C 180,E1 28331.944,E2 28331.944} C_VEL
LIN {X 0,Y 600.076,Z 1099.324,A -85,B 0,C 180,E1 28330.128,E2 28330.128} C_VEL
LIN {X 0,Y 600.16,Z 1083.192,A -85,B 0,C 180,E1 28328.191,E2 28328.191} C_VEL
LIN {X 0,Y 600.271,Z 1066.527,A -85,B 0,C 180,E1 28326.436,E2 28326.436} C_VEL
LIN {X 0,Y 600.35,Z 1048.788,A -85,B 0,C 180,E1 28324.816,E2 28324.816} C_VEL
LIN {X 0,Y 600.479,Z 1028.385,A -85,B 0,C 180,E1 28323.187,E2 28323.187} C_VEL
LIN {X 0,Y 600.599,Z 1008.93,A -85,B 0,C 180,E1 28321.838,E2 28321.838} C_VEL
LIN {X 0,Y 600.716,Z 988.803,A -85,B 0,C 180,E1 28320.647,E2 28320.647} C_VEL
LIN {X 0,Y 600.842,Z 967.727,A -85,B 0,C 180,E1 28319.574,E2 28319.574} C_VEL
LIN {X 0,Y 600.942,Z 946.648,A -85,B 0,C 180,E1 28318.699,E2 28318.699} C_VEL
LIN {X 0,Y 601.031,Z 925.495,A -85,B 0,C 180,E1 28317.975,E2 28317.975} C_VEL
LIN {X 0,Y 601.111,Z 903.411,A -85,B 0,C 180,E1 28317.41,E2 28317.41} C_VEL
LIN {X 0,Y 601.159,Z 883.61,A -85,B 0,C 180,E1 28317.041,E2 28317.041} C_VEL
LIN {X 0,Y 601.346,Z 675.485,A -85,B 0,C 180,E1 28314.092,E2 28314.092} C_VEL
LIN {X 0,Y 601.325,Z 543.956,A -85,B 0,C 180,E1 28312.167,E2 28312.167} C_VEL
LIN {X 0,Y 601.122,Z 542.023,A -85,B 0,C 180,E1 28312.077,E2 28312.077} C_VEL
LIN {X 0,Y 601.125,Z 511.56,A -85,B 0,C 180,E1 28309.991,E2 28309.991} C_VEL
LIN {X 0,Y 599.961,Z 508.314,A -85,B 0,C 180,E1 28309.653,E2 28309.653} C_VEL
LIN {X 0,Y 599.913,Z 508.316,A -85,B 0,C 180,E1 28306.607,E2 28306.607} C_VEL
LIN {X 0,Y 599.979,Z 508.31,A -85,B 0,C 180,E1 28303.492,E2 28303.492} C_VEL
LIN {X 0,Y 599.919,Z 508.313,A -85,B 0,C 180,E1 28300.388,E2 28300.388} C_VEL
LIN {X 0,Y 599.976,Z 508.311,A -85,B 0,C 180,E1 28297.224,E2 28297.224} C_VEL
LIN {X 0,Y 599.928,Z 508.311,A -85,B 0,C 180,E1 28294.055,E2 28294.055} C_VEL
LIN {X 0,Y 599.974,Z 508.308,A -85,B 0,C 180,E1 28290.882,E2 28290.882} C_VEL
LIN {X 0,Y 599.935,Z 508.311,A -85,B 0,C 180,E1 28287.751,E2 28287.751} C_VEL
LIN {X 0,Y 599.971,Z 508.306,A -85,B 0,C 180,E1 28284.622,E2 28284.622} C_VEL
LIN {X 0,Y 599.941,Z 508.311,A -85,B 0,C 180,E1 28281.509,E2 28281.509} C_VEL
LIN {X 0,Y 599.965,Z 508.306,A -85,B 0,C 180,E1 28278.359,E2 28278.359} C_VEL
LIN {X 0,Y 599.948,Z 508.31,A -85,B 0,C 180,E1 28275.213,E2 28275.213} C_VEL
LIN {X 0,Y 599.961,Z 508.308,A -85,B 0,C 180,E1 28272.121,E2 28272.121} C_VEL
LIN {X 0,Y 599.953,Z 508.308,A -85,B 0,C 180,E1 28269.013,E2 28269.013} C_VEL
LIN {X 0,Y 599.956,Z 508.31,A -85,B 0,C 180,E1 28265.835,E2 28265.835} C_VEL
LIN {X 0,Y 599.958,Z 508.31,A -85,B 0,C 180,E1 28262.674,E2 28262.674} C_VEL
LIN {X 0,Y 599.951,Z 508.31,A -85,B 0,C 180,E1 28259.522,E2 28259.522} C_VEL
LIN {X 0,Y 599.963,Z 508.311,A -85,B 0,C 180,E1 28256.369,E2 28256.369} C_VEL
LIN {X 0,Y 599.948,Z 508.313,A -85,B 0,C 180,E1 28253.433,E2 28253.433} C_VEL
LIN {X 0,Y 598.947,Z 508.437,A -85,B 0,C 180,E1 28252.697,E2 28252.697} C_VEL
LIN {X 0,Y 592.556,Z 509.229,A -85,B 0,C 180,E1 28250.633,E2 28250.633} C_VEL
LIN {X 0,Y 592.029,Z 509.297,A -85,B 0,C 180,E1 28250.096,E2 28250.096} C_VEL
LIN {X 0,Y 591.999,Z 509.3,A -85,B 0,C 180,E1 28246.919,E2 28246.919} C_VEL
LIN {X 0,Y 592.032,Z 509.3,A -85,B 0,C 180,E1 28243.719,E2 28243.719} C_VEL
LIN {X 0,Y 591.992,Z 509.3,A -85,B 0,C 180,E1 28240.565,E2 28240.565} C_VEL
LIN {X 0,Y 592.037,Z 509.303,A -85,B 0,C 180,E1 28237.353,E2 28237.353} C_VEL
LIN {X 0,Y 591.986,Z 509.3,A -85,B 0,C 180,E1 28234.19,E2 28234.19} C_VEL
LIN {X 0,Y 592.037,Z 509.301,A -85,B 0,C 180,E1 28231.007,E2 28231.007} C_VEL
LIN {X 0,Y 591.976,Z 509.302,A -85,B 0,C 180,E1 28227.971,E2 28227.971} C_VEL
LIN {X 0,Y 592.036,Z 509.3,A -85,B 0,C 180,E1 28224.826,E2 28224.826} C_VEL
LIN {X 0,Y 591.967,Z 509.302,A -85,B 0,C 180,E1 28221.759,E2 28221.759} C_VEL
LIN {X 0,Y 592.037,Z 509.302,A -85,B 0,C 180,E1 28218.674,E2 28218.674} C_VEL
LIN {X 0,Y 591.96,Z 509.305,A -85,B 0,C 180,E1 28215.601,E2 28215.601} C_VEL
LIN {X 0,Y 591.982,Z 509.3,A -85,B 0,C 180,E1 28212.764,E2 28212.764} C_VEL
LIN {X 0,Y 591.957,Z 509.31,A -85,B 0,C 180,E1 28209.475,E2 28209.475} C_VEL
LIN {X 0,Y 591.973,Z 509.435,A -85,B 0,C 180,E1 28208.802,E2 28208.802} C_VEL
LIN {X 0,Y 593.826,Z 513.93,A -85,B 0,C 180,E1 28208.352,E2 28208.352} C_VEL
LIN {X 0,Y 595.062,Z 516.901,A -85,B 0,C 180,E1 28208.213,E2 28208.213} C_VEL
LIN {X 0,Y 594.797,Z 669.548,A -85,B 0,C 180,E1 28205.968,E2 28205.968} C_VEL
LIN {X 0,Y 594.411,Z 861.423,A -85,B 0,C 180,E1 28203.205,E2 28203.205} C_VEL
LIN {X 0,Y 594.251,Z 885.144,A -85,B 0,C 180,E1 28202.68,E2 28202.68} C_VEL
LIN {X 0,Y 594.109,Z 905.38,A -85,B 0,C 180,E1 28202.072,E2 28202.072} C_VEL
LIN {X 0,Y 593.86,Z 928.521,A -85,B 0,C 180,E1 28201.186,E2 28201.186} C_VEL
LIN {X 0,Y 593.68,Z 948.815,A -85,B 0,C 180,E1 28200.234,E2 28200.234} C_VEL
LIN {X 0,Y 593.396,Z 970.575,A -85,B 0,C 180,E1 28199.014,E2 28199.014} C_VEL
LIN {X 0,Y 593.179,Z 991.069,A -85,B 0,C 180,E1 28197.671,E2 28197.671} C_VEL
LIN {X 0,Y 592.924,Z 1010.053,A -85,B 0,C 180,E1 28196.218,E2 28196.218} C_VEL
LIN {X 0,Y 592.677,Z 1029.431,A -85,B 0,C 180,E1 28194.52,E2 28194.52} C_VEL
LIN {X 0,Y 592.517,Z 1046.74,A -85,B 0,C 180,E1 28192.785,E2 28192.785} C_VEL
LIN {X 0,Y 592.34,Z 1062.468,A -85,B 0,C 180,E1 28190.969,E2 28190.969} C_VEL
LIN {X 0,Y 592.193,Z 1078.014,A -85,B 0,C 180,E1 28188.916,E2 28188.916} C_VEL
LIN {X 0,Y 592.114,Z 1090.73,A -85,B 0,C 180,E1 28186.986,E2 28186.986} C_VEL
LIN {X 0,Y 592.033,Z 1102.078,A -85,B 0,C 180,E1 28184.975,E2 28184.975} C_VEL
LIN {X 0,Y 591.974,Z 1111.941,A -85,B 0,C 180,E1 28182.95,E2 28182.95} C_VEL
LIN {X 0,Y 591.939,Z 1120.529,A -85,B 0,C 180,E1 28180.807,E2 28180.807} C_VEL
LIN {X 0,Y 591.93,Z 1127.336,A -85,B 0,C 180,E1 28178.744,E2 28178.744} C_VEL
LIN {X 0,Y 591.913,Z 1132.951,A -85,B 0,C 180,E1 28176.499,E2 28176.499} C_VEL
LIN {X 0,Y 591.91,Z 1136.838,A -85,B 0,C 180,E1 28174.36,E2 28174.36} C_VEL
LIN {X 0,Y 591.916,Z 1139.157,A -85,B 0,C 180,E1 28172.13,E2 28172.13} C_VEL
LIN {X 0,Y 591.911,Z 1139.996,A -85,B 0,C 180,E1 28170,E2 28170} C_VEL
LIN {X 0,Y 591.915,Z 1139.22,A -85,B 0,C 180,E1 28167.87,E2 28167.87} C_VEL
LIN {X 0,Y 591.909,Z 1136.982,A -85,B 0,C 180,E1 28165.641,E2 28165.641} C_VEL
LIN {X 0,Y 591.92,Z 1133.143,A -85,B 0,C 180,E1 28163.502,E2 28163.502} C_VEL
LIN {X 0,Y 591.929,Z 1127.901,A -85,B 0,C 180,E1 28161.354,E2 28161.354} C_VEL
LIN {X 0,Y 591.937,Z 1120.856,A -85,B 0,C 180,E1 28159.194,E2 28159.194} C_VEL
LIN {X 0,Y 591.979,Z 1112.346,A -85,B 0,C 180,E1 28157.048,E2 28157.048} C_VEL
LIN {X 0,Y 592.031,Z 1102.536,A -85,B 0,C 180,E1 28155.023,E2 28155.023} C_VEL
LIN {X 0,Y 592.116,Z 1090.662,A -85,B 0,C 180,E1 28152.913,E2 28152.913} C_VEL
LIN {X 0,Y 592.196,Z 1077.932,A -85,B 0,C 180,E1 28150.982,E2 28150.982} C_VEL
LIN {X 0,Y 592.343,Z 1062.36,A -85,B 0,C 180,E1 28148.928,E2 28148.928} C_VEL
LIN {X 0,Y 592.517,Z 1046.754,A -85,B 0,C 180,E1 28147.126,E2 28147.126} C_VEL
LIN {X 0,Y 592.679,Z 1029.266,A -85,B 0,C 180,E1 28145.374,E2 28145.374} C_VEL
LIN {X 0,Y 592.926,Z 1009.811,A -85,B 0,C 180,E1 28143.673,E2 28143.673} C_VEL
LIN {X 0,Y 593.179,Z 991.129,A -85,B 0,C 180,E1 28142.244,E2 28142.244} C_VEL
LIN {X 0,Y 593.395,Z 970.869,A -85,B 0,C 180,E1 28140.914,E2 28140.914} C_VEL
LIN {X 0,Y 593.676,Z 949.444,A -85,B 0,C 180,E1 28139.708,E2 28139.708} C_VEL
LIN {X 0,Y 593.855,Z 929.417,A -85,B 0,C 180,E1 28138.764,E2 28138.764} C_VEL
LIN {X 0,Y 594.102,Z 906.827,A -85,B 0,C 180,E1 28137.886,E2 28137.886} C_VEL
LIN {X 0,Y 594.247,Z 886.165,A -85,B 0,C 180,E1 28137.258,E2 28137.258} C_VEL
LIN {X 0,Y 594.407,Z 863.614,A -85,B 0,C 180,E1 28136.742,E2 28136.742} C_VEL
LIN {X 0,Y 594.537,Z 811.969,A -85,B 0,C 180,E1 28135.981,E2 28135.981} C_VEL
LIN {X 0,Y 595,Z 599.474,A -85,B 0,C 180,E1 28132.925,E2 28132.925} C_VEL
LIN {X 0,Y 594.949,Z 516.352,A -85,B 0,C 180,E1 28131.68,E2 28131.68} C_VEL
LIN {X 0,Y 593.474,Z 513.051,A -85,B 0,C 180,E1 28131.496,E2 28131.496} C_VEL
LIN {X 0,Y 592.014,Z 509.71,A -85,B 0,C 180,E1 28131.132,E2 28131.132} C_VEL
LIN {X 0,Y 591.95,Z 509.31,A -85,B 0,C 180,E1 28131.072,E2 28131.072} C_VEL
LIN {X 0,Y 591.96,Z 509.308,A -85,B 0,C 180,E1 28128.28,E2 28128.28} C_VEL
LIN {X 0,Y 591.964,Z 509.306,A -85,B 0,C 180,E1 28124.912,E2 28124.912} C_VEL
LIN {X 0,Y 591.961,Z 509.305,A -85,B 0,C 180,E1 28122.141,E2 28122.141} C_VEL
LIN {X 0,Y 592.003,Z 509.301,A -85,B 0,C 180,E1 28118.924,E2 28118.924} C_VEL
LIN {X 0,Y 591.965,Z 509.304,A -85,B 0,C 180,E1 28115.996,E2 28115.996} C_VEL
LIN {X 0,Y 592.039,Z 509.3,A -85,B 0,C 180,E1 28112.828,E2 28112.828} C_VEL
LIN {X 0,Y 591.974,Z 509.3,A -85,B 0,C 180,E1 28109.754,E2 28109.754} C_VEL
LIN {X 0,Y 592.039,Z 509.302,A -85,B 0,C 180,E1 28106.695,E2 28106.695} C_VEL
LIN {X 0,Y 591.981,Z 509.297,A -85,B 0,C 180,E1 28103.597,E2 28103.597} C_VEL
LIN {X 0,Y 592.037,Z 509.304,A -85,B 0,C 180,E1 28100.566,E2 28100.566} C_VEL
LIN {X 0,Y 591.991,Z 509.295,A -85,B 0,C 180,E1 28097.394,E2 28097.394} C_VEL
LIN {X 0,Y 592.034,Z 509.304,A -85,B 0,C 180,E1 28094.275,E2 28094.275} C_VEL
LIN {X 0,Y 592,Z 509.298,A -85,B 0,C 180,E1 28091.101,E2 28091.101} C_VEL
LIN {X 0,Y 592.033,Z 509.302,A -85,B 0,C 180,E1 28087.96,E2 28087.96} C_VEL
LIN {X 0,Y 592.005,Z 509.298,A -85,B 0,C 180,E1 28084.747,E2 28084.747} C_VEL
LIN {X 0,Y 592.027,Z 509.3,A -85,B 0,C 180,E1 28081.645,E2 28081.645} C_VEL
LIN {X 0,Y 592.012,Z 509.298,A -85,B 0,C 180,E1 28078.452,E2 28078.452} C_VEL
LIN {X 0,Y 592.022,Z 509.301,A -85,B 0,C 180,E1 28075.35,E2 28075.35} C_VEL
LIN {X 0,Y 592.018,Z 509.298,A -85,B 0,C 180,E1 28072.137,E2 28072.137} C_VEL
LIN {X 0,Y 592.016,Z 509.295,A -85,B 0,C 180,E1 28068.998,E2 28068.998} C_VEL
LIN {X 0,Y 592.022,Z 509.299,A -85,B 0,C 180,E1 28065.795,E2 28065.795} C_VEL
LIN {X 0,Y 592.007,Z 509.294,A -85,B 0,C 180,E1 28062.606,E2 28062.606} C_VEL
LIN {X 0,Y 592.027,Z 509.3,A -85,B 0,C 180,E1 28059.434,E2 28059.434} C_VEL
LIN {X 0,Y 592.001,Z 509.296,A -85,B 0,C 180,E1 28056.299,E2 28056.299} C_VEL
LIN {X 0,Y 592.03,Z 509.302,A -85,B 0,C 180,E1 28053.089,E2 28053.089} C_VEL
LIN {X 0,Y 591.993,Z 509.299,A -85,B 0,C 180,E1 28050.005,E2 28050.005} C_VEL
LIN {X 0,Y 592.035,Z 509.301,A -85,B 0,C 180,E1 28046.826,E2 28046.826} C_VEL
LIN {X 0,Y 591.987,Z 509.301,A -85,B 0,C 180,E1 28043.673,E2 28043.673} C_VEL
LIN {X 0,Y 592.037,Z 509.301,A -85,B 0,C 180,E1 28040.455,E2 28040.455} C_VEL
LIN {X 0,Y 591.979,Z 509.301,A -85,B 0,C 180,E1 28037.368,E2 28037.368} C_VEL
LIN {X 0,Y 592.04,Z 509.304,A -85,B 0,C 180,E1 28034.226,E2 28034.226} C_VEL
LIN {X 0,Y 591.969,Z 509.308,A -85,B 0,C 180,E1 28031.123,E2 28031.123} C_VEL
LIN {X 0,Y 591.995,Z 509.462,A -85,B 0,C 180,E1 28030.904,E2 28030.904} C_VEL
LIN {X 0,Y 593.39,Z 512.911,A -85,B 0,C 180,E1 28030.542,E2 28030.542} C_VEL
LIN {X 0,Y 594.606,Z 516.07,A -85,B 0,C 180,E1 28030.219,E2 28030.219} C_VEL
LIN {X 0,Y 594.516,Z 543.463,A -85,B 0,C 180,E1 28028.352,E2 28028.352} C_VEL
LIN {X 0,Y 595.158,Z 547.745,A -85,B 0,C 180,E1 28028.238,E2 28028.238} C_VEL
LIN {X 0,Y 594.756,Z 726.838,A -85,B 0,C 180,E1 28025.618,E2 28025.618} C_VEL
LIN {X 0,Y 594.412,Z 891.453,A -85,B 0,C 180,E1 28023.249,E2 28023.249} C_VEL
LIN {X 0,Y 594.252,Z 915.121,A -85,B 0,C 180,E1 28022.726,E2 28022.726} C_VEL
LIN {X 0,Y 594.109,Z 935.358,A -85,B 0,C 180,E1 28022.117,E2 28022.117} C_VEL
LIN {X 0,Y 593.861,Z 958.402,A -85,B 0,C 180,E1 28021.236,E2 28021.236} C_VEL
LIN {X 0,Y 593.682,Z 978.543,A -85,B 0,C 180,E1 28020.292,E2 28020.292} C_VEL
LIN {X 0,Y 593.399,Z 1000.144,A -85,B 0,C 180,E1 28019.085,E2 28019.085} C_VEL
LIN {X 0,Y 593.194,Z 1020.453,A -85,B 0,C 180,E1 28017.76,E2 28017.76} C_VEL
LIN {X 0,Y 592.93,Z 1039.258,A -85,B 0,C 180,E1 28016.327,E2 28016.327} C_VEL
LIN {X 0,Y 592.699,Z 1058.325,A -85,B 0,C 180,E1 28014.67,E2 28014.67} C_VEL
LIN {X 0,Y 592.524,Z 1075.351,A -85,B 0,C 180,E1 28012.975,E2 28012.975} C_VEL
LIN {X 0,Y 592.349,Z 1091.138,A -85,B 0,C 180,E1 28011.175,E2 28011.175} C_VEL
LIN {X 0,Y 592.236,Z 1105.582,A -85,B 0,C 180,E1 28009.311,E2 28009.311} C_VEL
LIN {X 0,Y 592.125,Z 1118.45,A -85,B 0,C 180,E1 28007.39,E2 28007.39} C_VEL
LIN {X 0,Y 592.031,Z 1130.751,A -85,B 0,C 180,E1 28005.275,E2 28005.275} C_VEL
LIN {X 0,Y 591.963,Z 1140.184,A -85,B 0,C 180,E1 28003.372,E2 28003.372} C_VEL
LIN {X 0,Y 591.935,Z 1149.269,A -85,B 0,C 180,E1 28001.201,E2 28001.201} C_VEL
LIN {X 0,Y 591.918,Z 1155.954,A -85,B 0,C 180,E1 27999.234,E2 27999.234} C_VEL
LIN {X 0,Y 591.888,Z 1161.807,A -85,B 0,C 180,E1 27997.083,E2 27997.083} C_VEL
LIN {X 0,Y 591.907,Z 1165.957,A -85,B 0,C 180,E1 27994.942,E2 27994.942} C_VEL
LIN {X 0,Y 591.896,Z 1168.718,A -85,B 0,C 180,E1 27992.808,E2 27992.808} C_VEL
LIN {X 0,Y 591.882,Z 1169.85,A -85,B 0,C 180,E1 27990.677,E2 27990.677} C_VEL
LIN {X 0,Y 591.91,Z 1169.657,A -85,B 0,C 180,E1 27988.548,E2 27988.548} C_VEL
LIN {X 0,Y 591.894,Z 1167.84,A -85,B 0,C 180,E1 27986.416,E2 27986.416} C_VEL
LIN {X 0,Y 591.89,Z 1164.629,A -85,B 0,C 180,E1 27984.25,E2 27984.25} C_VEL
LIN {X 0,Y 591.921,Z 1159.824,A -85,B 0,C 180,E1 27982.136,E2 27982.136} C_VEL
LIN {X 0,Y 591.912,Z 1153.818,A -85,B 0,C 180,E1 27980.078,E2 27980.078} C_VEL
LIN {X 0,Y 591.939,Z 1145.74,A -85,B 0,C 180,E1 27977.909,E2 27977.909} C_VEL
LIN {X 0,Y 592.004,Z 1136.9,A -85,B 0,C 180,E1 27975.924,E2 27975.924} C_VEL
LIN {X 0,Y 592.06,Z 1125.714,A -85,B 0,C 180,E1 27973.82,E2 27973.82} C_VEL
LIN {X 0,Y 592.157,Z 1113.276,A -85,B 0,C 180,E1 27971.797,E2 27971.797} C_VEL
LIN {X 0,Y 592.259,Z 1099.325,A -85,B 0,C 180,E1 27969.855,E2 27969.855} C_VEL
LIN {X 0,Y 592.433,Z 1082.727,A -85,B 0,C 180,E1 27967.839,E2 27967.839} C_VEL
LIN {X 0,Y 592.639,Z 1066.527,A -85,B 0,C 180,E1 27966.114,E2 27966.114} C_VEL
LIN {X 0,Y 592.806,Z 1048.751,A -85,B 0,C 180,E1 27964.469,E2 27964.469} C_VEL
LIN {X 0,Y 593.065,Z 1029.301,A -85,B 0,C 180,E1 27962.893,E2 27962.893} C_VEL
LIN {X 0,Y 593.283,Z 1010.55,A -85,B 0,C 180,E1 27961.569,E2 27961.569} C_VEL
LIN {X 0,Y 593.537,Z 989.801,A -85,B 0,C 180,E1 27960.312,E2 27960.312} C_VEL
LIN {X 0,Y 593.756,Z 969.575,A -85,B 0,C 180,E1 27959.264,E2 27959.264} C_VEL
LIN {X 0,Y 593.99,Z 947.385,A -85,B 0,C 180,E1 27958.319,E2 27958.319} C_VEL
LIN {X 0,Y 594.178,Z 925.959,A -85,B 0,C 180,E1 27957.576,E2 27957.576} C_VEL
LIN {X 0,Y 594.338,Z 903.575,A -85,B 0,C 180,E1 27956.995,E2 27956.995} C_VEL
LIN {X 0,Y 594.436,Z 883.289,A -85,B 0,C 180,E1 27956.615,E2 27956.615} C_VEL
LIN {X 0,Y 594.853,Z 678.196,A -85,B 0,C 180,E1 27953.678,E2 27953.678} C_VEL
LIN {X 0,Y 595.002,Z 545.703,A -85,B 0,C 180,E1 27951.719,E2 27951.719} C_VEL
LIN {X 0,Y 594.411,Z 542.656,A -85,B 0,C 180,E1 27951.615,E2 27951.615} C_VEL
LIN {X 0,Y 594.417,Z 515.332,A -85,B 0,C 180,E1 27949.713,E2 27949.713} C_VEL
LIN {X 0,Y 591.995,Z 509.461,A -85,B 0,C 180,E1 27949.096,E2 27949.096} C_VEL
LIN {X 0,Y 592.006,Z 509.304,A -85,B 0,C 180,E1 27946.151,E2 27946.151} C_VEL
LIN {X 0,Y 591.985,Z 509.301,A -85,B 0,C 180,E1 27942.859,E2 27942.859} C_VEL
LIN {X 0,Y 592.023,Z 509.306,A -85,B 0,C 180,E1 27939.785,E2 27939.785} C_VEL
LIN {X 0,Y 591.99,Z 509.301,A -85,B 0,C 180,E1 27936.49,E2 27936.49} C_VEL
LIN {X 0,Y 592.035,Z 509.301,A -85,B 0,C 180,E1 27933.405,E2 27933.405} C_VEL
LIN {X 0,Y 591.994,Z 509.298,A -85,B 0,C 180,E1 27930.145,E2 27930.145} C_VEL
LIN {X 0,Y 592.035,Z 509.303,A -85,B 0,C 180,E1 27927.02,E2 27927.02} C_VEL
LIN {X 0,Y 592.002,Z 509.294,A -85,B 0,C 180,E1 27923.807,E2 27923.807} C_VEL
LIN {X 0,Y 592.031,Z 509.301,A -85,B 0,C 180,E1 27920.668,E2 27920.668} C_VEL
LIN {X 0,Y 592.008,Z 509.293,A -85,B 0,C 180,E1 27917.495,E2 27917.495} C_VEL
LIN {X 0,Y 592.026,Z 509.302,A -85,B 0,C 180,E1 27914.375,E2 27914.375} C_VEL
LIN {X 0,Y 592.014,Z 509.294,A -85,B 0,C 180,E1 27911.199,E2 27911.199} C_VEL
LIN {X 0,Y 592.021,Z 509.301,A -85,B 0,C 180,E1 27908.058,E2 27908.058} C_VEL
LIN {X 0,Y 592.019,Z 509.298,A -85,B 0,C 180,E1 27904.823,E2 27904.823} C_VEL
LIN {X 0,Y 592.013,Z 509.299,A -85,B 0,C 180,E1 27901.645,E2 27901.645} C_VEL
LIN {X 0,Y 592.024,Z 509.298,A -85,B 0,C 180,E1 27898.548,E2 27898.548} C_VEL
LIN {X 0,Y 592.009,Z 509.3,A -85,B 0,C 180,E1 27895.447,E2 27895.447} C_VEL
LIN {X 0,Y 592.028,Z 509.299,A -85,B 0,C 180,E1 27892.235,E2 27892.235} C_VEL
LIN {X 0,Y 592.029,Z 509.297,A -85,B 0,C 180,E1 27890.096,E2 27890.096} C_VEL
LIN {X 0,Y 591.033,Z 509.428,A -85,B 0,C 180,E1 27889.35,E2 27889.35} C_VEL
LIN {X 0,Y 584.582,Z 510.228,A -85,B 0,C 180,E1 27887.259,E2 27887.259} C_VEL
LIN {X 0,Y 584.065,Z 510.287,A -85,B 0,C 180,E1 27886.714,E2 27886.714} C_VEL
LIN {X 0,Y 584.093,Z 510.286,A -85,B 0,C 180,E1 27883.389,E2 27883.389} C_VEL
LIN {X 0,Y 584.071,Z 510.286,A -85,B 0,C 180,E1 27880.187,E2 27880.187} C_VEL
LIN {X 0,Y 584.061,Z 510.284,A -85,B 0,C 180,E1 27876.813,E2 27876.813} C_VEL
LIN {X 0,Y 584.082,Z 510.287,A -85,B 0,C 180,E1 27873.681,E2 27873.681} C_VEL
LIN {X 0,Y 584.046,Z 510.288,A -85,B 0,C 180,E1 27870.422,E2 27870.422} C_VEL
LIN {X 0,Y 584.076,Z 510.289,A -85,B 0,C 180,E1 27867.368,E2 27867.368} C_VEL
LIN {X 0,Y 584.041,Z 510.293,A -85,B 0,C 180,E1 27864.162,E2 27864.162} C_VEL
LIN {X 0,Y 584.056,Z 510.289,A -85,B 0,C 180,E1 27861.163,E2 27861.163} C_VEL
LIN {X 0,Y 584.031,Z 510.294,A -85,B 0,C 180,E1 27857.843,E2 27857.843} C_VEL
LIN {X 0,Y 584.036,Z 510.294,A -85,B 0,C 180,E1 27854.996,E2 27854.996} C_VEL
LIN {X 0,Y 584.026,Z 510.298,A -85,B 0,C 180,E1 27851.626,E2 27851.626} C_VEL
LIN {X 0,Y 584.033,Z 510.456,A -85,B 0,C 180,E1 27849.354,E2 27849.354} C_VEL
LIN {X 0,Y 585.438,Z 513.958,A -85,B 0,C 180,E1 27849.005,E2 27849.005} C_VEL
LIN {X 0,Y 588.827,Z 519.669,A -85,B 0,C 180,E1 27848.651,E2 27848.651} C_VEL
LIN {X 0,Y 588.256,Z 692.998,A -85,B 0,C 180,E1 27846.085,E2 27846.085} C_VEL
LIN {X 0,Y 587.709,Z 861.574,A -85,B 0,C 180,E1 27843.632,E2 27843.632} C_VEL
LIN {X 0,Y 587.465,Z 885.432,A -85,B 0,C 180,E1 27843.098,E2 27843.098} C_VEL
LIN {X 0,Y 587.248,Z 906.266,A -85,B 0,C 180,E1 27842.463,E2 27842.463} C_VEL
LIN {X 0,Y 586.878,Z 928.818,A -85,B 0,C 180,E1 27841.587,E2 27841.587} C_VEL
LIN {X 0,Y 586.595,Z 949.661,A -85,B 0,C 180,E1 27840.596,E2 27840.596} C_VEL
LIN {X 0,Y 586.181,Z 970.315,A -85,B 0,C 180,E1 27839.423,E2 27839.423} C_VEL
LIN {X 0,Y 585.864,Z 990.696,A -85,B 0,C 180,E1 27838.075,E2 27838.075} C_VEL
LIN {X 0,Y 585.463,Z 1010.032,A -85,B 0,C 180,E1 27836.58,E2 27836.58} C_VEL
LIN {X 0,Y 585.11,Z 1029.504,A -85,B 0,C 180,E1 27834.852,E2 27834.852} C_VEL
LIN {X 0,Y 584.843,Z 1046.699,A -85,B 0,C 180,E1 27833.107,E2 27833.107} C_VEL
LIN {X 0,Y 584.57,Z 1062.781,A -85,B 0,C 180,E1 27831.223,E2 27831.223} C_VEL
LIN {X 0,Y 584.356,Z 1078.023,A -85,B 0,C 180,E1 27829.179,E2 27829.179} C_VEL
LIN {X 0,Y 584.225,Z 1090.732,A -85,B 0,C 180,E1 27827.222,E2 27827.222} C_VEL
LIN {X 0,Y 584.093,Z 1102.604,A -85,B 0,C 180,E1 27825.082,E2 27825.082} C_VEL
LIN {X 0,Y 584.009,Z 1112.694,A -85,B 0,C 180,E1 27822.961,E2 27822.961} C_VEL
LIN {X 0,Y 583.954,Z 1120.888,A -85,B 0,C 180,E1 27820.856,E2 27820.856} C_VEL
LIN {X 0,Y 583.938,Z 1127.923,A -85,B 0,C 180,E1 27818.667,E2 27818.667} C_VEL
LIN {X 0,Y 583.915,Z 1133.159,A -85,B 0,C 180,E1 27816.489,E2 27816.489} C_VEL
LIN {X 0,Y 583.916,Z 1137.111,A -85,B 0,C 180,E1 27814.223,E2 27814.223} C_VEL
LIN {X 0,Y 583.913,Z 1139.225,A -85,B 0,C 180,E1 27812.061,E2 27812.061} C_VEL
LIN {X 0,Y 583.903,Z 1139.972,A -85,B 0,C 180,E1 27809.804,E2 27809.804} C_VEL
LIN {X 0,Y 583.916,Z 1139.153,A -85,B 0,C 180,E1 27807.743,E2 27807.743} C_VEL
LIN {X 0,Y 583.902,Z 1136.827,A -85,B 0,C 180,E1 27805.482,E2 27805.482} C_VEL
LIN {X 0,Y 583.905,Z 1132.908,A -85,B 0,C 180,E1 27803.301,E2 27803.301} C_VEL
LIN {X 0,Y 583.938,Z 1127.311,A -85,B 0,C 180,E1 27801.036,E2 27801.036} C_VEL
LIN {X 0,Y 583.948,Z 1120.499,A -85,B 0,C 180,E1 27798.944,E2 27798.944} C_VEL
LIN {X 0,Y 584.002,Z 1111.746,A -85,B 0,C 180,E1 27796.737,E2 27796.737} C_VEL
LIN {X 0,Y 584.091,Z 1102.025,A -85,B 0,C 180,E1 27794.715,E2 27794.715} C_VEL
LIN {X 0,Y 584.228,Z 1090.019,A -85,B 0,C 180,E1 27792.573,E2 27792.573} C_VEL
LIN {X 0,Y 584.376,Z 1077.221,A -85,B 0,C 180,E1 27790.614,E2 27790.614} C_VEL
LIN {X 0,Y 584.58,Z 1062.355,A -85,B 0,C 180,E1 27788.635,E2 27788.635} C_VEL
LIN {X 0,Y 584.845,Z 1046.613,A -85,B 0,C 180,E1 27786.794,E2 27786.794} C_VEL
LIN {X 0,Y 585.117,Z 1029.259,A -85,B 0,C 180,E1 27785.034,E2 27785.034} C_VEL
LIN {X 0,Y 585.466,Z 1009.804,A -85,B 0,C 180,E1 27783.311,E2 27783.311} C_VEL
LIN {X 0,Y 585.862,Z 990.807,A -85,B 0,C 180,E1 27781.843,E2 27781.843} C_VEL
LIN {X 0,Y 586.174,Z 970.861,A -85,B 0,C 180,E1 27780.521,E2 27780.521} C_VEL
LIN {X 0,Y 586.597,Z 949.433,A -85,B 0,C 180,E1 27779.303,E2 27779.303} C_VEL
LIN {X 0,Y 586.871,Z 929.404,A -85,B 0,C 180,E1 27778.349,E2 27778.349} C_VEL
LIN {X 0,Y 587.245,Z 906.485,A -85,B 0,C 180,E1 27777.454,E2 27777.454} C_VEL
LIN {X 0,Y 587.463,Z 885.712,A -85,B 0,C 180,E1 27776.819,E2 27776.819} C_VEL
LIN {X 0,Y 587.707,Z 862.397,A -85,B 0,C 180,E1 27776.292,E2 27776.292} C_VEL
LIN {X 0,Y 587.979,Z 786.94,A -85,B 0,C 180,E1 27775.186,E2 27775.186} C_VEL
LIN {X 0,Y 588.654,Z 572.392,A -85,B 0,C 180,E1 27772.049,E2 27772.049} C_VEL
LIN {X 0,Y 588.705,Z 519.198,A -85,B 0,C 180,E1 27771.242,E2 27771.242} C_VEL
LIN {X 0,Y 584.889,Z 513.084,A -85,B 0,C 180,E1 27770.828,E2 27770.828} C_VEL
LIN {X 0,Y 584.012,Z 510.301,A -85,B 0,C 180,E1 27770.525,E2 27770.525} C_VEL
LIN {X 0,Y 584.044,Z 510.297,A -85,B 0,C 180,E1 27767.259,E2 27767.259} C_VEL
LIN {X 0,Y 584.012,Z 510.296,A -85,B 0,C 180,E1 27764.445,E2 27764.445} C_VEL
LIN {X 0,Y 584.096,Z 510.292,A -85,B 0,C 180,E1 27761.281,E2 27761.281} C_VEL
LIN {X 0,Y 584.022,Z 510.291,A -85,B 0,C 180,E1 27758.173,E2 27758.173} C_VEL
LIN {X 0,Y 584.098,Z 510.286,A -85,B 0,C 180,E1 27755.091,E2 27755.091} C_VEL
LIN {X 0,Y 584.033,Z 510.292,A -85,B 0,C 180,E1 27752.054,E2 27752.054} C_VEL
LIN {X 0,Y 584.093,Z 510.287,A -85,B 0,C 180,E1 27748.976,E2 27748.976} C_VEL
LIN {X 0,Y 584.043,Z 510.29,A -85,B 0,C 180,E1 27745.775,E2 27745.775} C_VEL
LIN {X 0,Y 584.1,Z 510.288,A -85,B 0,C 180,E1 27742.653,E2 27742.653} C_VEL
LIN {X 0,Y 584.051,Z 510.289,A -85,B 0,C 180,E1 27739.501,E2 27739.501} C_VEL
LIN {X 0,Y 584.099,Z 510.287,A -85,B 0,C 180,E1 27736.406,E2 27736.406} C_VEL
LIN {X 0,Y 584.058,Z 510.289,A -85,B 0,C 180,E1 27733.161,E2 27733.161} C_VEL
LIN {X 0,Y 584.094,Z 510.291,A -85,B 0,C 180,E1 27730.056,E2 27730.056} C_VEL
LIN {X 0,Y 584.065,Z 510.288,A -85,B 0,C 180,E1 27726.831,E2 27726.831} C_VEL
LIN {X 0,Y 584.089,Z 510.289,A -85,B 0,C 180,E1 27723.627,E2 27723.627} C_VEL
LIN {X 0,Y 584.071,Z 510.287,A -85,B 0,C 180,E1 27720.393,E2 27720.393} C_VEL
LIN {X 0,Y 584.085,Z 510.286,A -85,B 0,C 180,E1 27717.155,E2 27717.155} C_VEL
LIN {X 0,Y 584.082,Z 510.291,A -85,B 0,C 180,E1 27713.908,E2 27713.908} C_VEL
LIN {X 0,Y 584.089,Z 510.283,A -85,B 0,C 180,E1 27710.641,E2 27710.641} C_VEL
LIN {X 0,Y 584.09,Z 510.292,A -85,B 0,C 180,E1 27707.243,E2 27707.243} C_VEL
LIN {X 0,Y 584.096,Z 510.283,A -85,B 0,C 180,E1 27704.002,E2 27704.002} C_VEL
LIN {X 0,Y 584.072,Z 510.29,A -85,B 0,C 180,E1 27700.708,E2 27700.708} C_VEL
LIN {X 0,Y 584.091,Z 510.286,A -85,B 0,C 180,E1 27697.559,E2 27697.559} C_VEL
LIN {X 0,Y 584.063,Z 510.291,A -85,B 0,C 180,E1 27694.335,E2 27694.335} C_VEL
LIN {X 0,Y 584.094,Z 510.286,A -85,B 0,C 180,E1 27691.136,E2 27691.136} C_VEL
LIN {X 0,Y 584.054,Z 510.29,A -85,B 0,C 180,E1 27687.948,E2 27687.948} C_VEL
LIN {X 0,Y 584.098,Z 510.287,A -85,B 0,C 180,E1 27684.739,E2 27684.739} C_VEL
LIN {X 0,Y 584.045,Z 510.287,A -85,B 0,C 180,E1 27681.579,E2 27681.579} C_VEL
LIN {X 0,Y 584.098,Z 510.289,A -85,B 0,C 180,E1 27678.381,E2 27678.381} C_VEL
LIN {X 0,Y 584.038,Z 510.292,A -85,B 0,C 180,E1 27675.273,E2 27675.273} C_VEL
LIN {X 0,Y 584.097,Z 510.294,A -85,B 0,C 180,E1 27672.146,E2 27672.146} C_VEL
LIN {X 0,Y 584.068,Z 510.48,A -85,B 0,C 180,E1 27671.507,E2 27671.507} C_VEL
LIN {X 0,Y 585.449,Z 513.943,A -85,B 0,C 180,E1 27671.136,E2 27671.136} C_VEL
LIN {X 0,Y 587.991,Z 519.651,A -85,B 0,C 180,E1 27670.51,E2 27670.51} C_VEL
LIN {X 0,Y 587.865,Z 543.525,A -85,B 0,C 180,E1 27668.865,E2 27668.865} C_VEL
LIN {X 0,Y 588.861,Z 549.34,A -85,B 0,C 180,E1 27668.698,E2 27668.698} C_VEL
LIN {X 0,Y 588.243,Z 728.619,A -85,B 0,C 180,E1 27666.047,E2 27666.047} C_VEL
LIN {X 0,Y 587.711,Z 891.56,A -85,B 0,C 180,E1 27663.677,E2 27663.677} C_VEL
LIN {X 0,Y 587.466,Z 915.293,A -85,B 0,C 180,E1 27663.147,E2 27663.147} C_VEL
LIN {X 0,Y 587.249,Z 936.007,A -85,B 0,C 180,E1 27662.517,E2 27662.517} C_VEL
LIN {X 0,Y 586.874,Z 959.128,A -85,B 0,C 180,E1 27661.618,E2 27661.618} C_VEL
LIN {X 0,Y 586.588,Z 980.558,A -85,B 0,C 180,E1 27660.596,E2 27660.596} C_VEL
LIN {X 0,Y 586.171,Z 1001.037,A -85,B 0,C 180,E1 27659.423,E2 27659.423} C_VEL
LIN {X 0,Y 585.845,Z 1021.343,A -85,B 0,C 180,E1 27658.072,E2 27658.072} C_VEL
LIN {X 0,Y 585.458,Z 1040.584,A -85,B 0,C 180,E1 27656.58,E2 27656.58} C_VEL
LIN {X 0,Y 585.096,Z 1059.99,A -85,B 0,C 180,E1 27654.85,E2 27654.85} C_VEL
LIN {X 0,Y 584.833,Z 1077.117,A -85,B 0,C 180,E1 27653.106,E2 27653.106} C_VEL
LIN {X 0,Y 584.568,Z 1093.14,A -85,B 0,C 180,E1 27651.224,E2 27651.224} C_VEL
LIN {X 0,Y 584.351,Z 1108.331,A -85,B 0,C 180,E1 27649.179,E2 27649.179} C_VEL
LIN {X 0,Y 584.216,Z 1121.645,A -85,B 0,C 180,E1 27647.12,E2 27647.12} C_VEL
LIN {X 0,Y 584.091,Z 1132.836,A -85,B 0,C 180,E1 27645.082,E2 27645.082} C_VEL
LIN {X 0,Y 584.008,Z 1142.879,A -85,B 0,C 180,E1 27642.96,E2 27642.96} C_VEL
LIN {X 0,Y 583.953,Z 1151.051,A -85,B 0,C 180,E1 27640.856,E2 27640.856} C_VEL
LIN {X 0,Y 583.936,Z 1158.04,A -85,B 0,C 180,E1 27638.666,E2 27638.666} C_VEL
LIN {X 0,Y 583.919,Z 1163.254,A -85,B 0,C 180,E1 27636.489,E2 27636.489} C_VEL
LIN {X 0,Y 583.916,Z 1167.164,A -85,B 0,C 180,E1 27634.222,E2 27634.222} C_VEL
LIN {X 0,Y 583.913,Z 1169.256,A -85,B 0,C 180,E1 27632.061,E2 27632.061} C_VEL
LIN {X 0,Y 583.9,Z 1169.962,A -85,B 0,C 180,E1 27629.804,E2 27629.804} C_VEL
LIN {X 0,Y 583.916,Z 1169.122,A -85,B 0,C 180,E1 27627.743,E2 27627.743} C_VEL
LIN {X 0,Y 583.904,Z 1166.753,A -85,B 0,C 180,E1 27625.482,E2 27625.482} C_VEL
LIN {X 0,Y 583.913,Z 1163.046,A -85,B 0,C 180,E1 27623.412,E2 27623.412} C_VEL
LIN {X 0,Y 583.936,Z 1157.774,A -85,B 0,C 180,E1 27621.234,E2 27621.234} C_VEL
LIN {X 0,Y 583.951,Z 1150.693,A -85,B 0,C 180,E1 27619.044,E2 27619.044} C_VEL
LIN {X 0,Y 584.005,Z 1142.455,A -85,B 0,C 180,E1 27616.938,E2 27616.938} C_VEL
LIN {X 0,Y 584.092,Z 1132.314,A -85,B 0,C 180,E1 27614.816,E2 27614.816} C_VEL
LIN {X 0,Y 584.226,Z 1120.376,A -85,B 0,C 180,E1 27612.675,E2 27612.675} C_VEL
LIN {X 0,Y 584.367,Z 1107.619,A -85,B 0,C 180,E1 27610.717,E2 27610.717} C_VEL
LIN {X 0,Y 584.571,Z 1092.839,A -85,B 0,C 180,E1 27608.739,E2 27608.739} C_VEL
LIN {X 0,Y 584.842,Z 1076.671,A -85,B 0,C 180,E1 27606.845,E2 27606.845} C_VEL
LIN {X 0,Y 585.098,Z 1059.899,A -85,B 0,C 180,E1 27605.141,E2 27605.141} C_VEL
LIN {X 0,Y 585.457,Z 1040.577,A -85,B 0,C 180,E1 27603.419,E2 27603.419} C_VEL
LIN {X 0,Y 585.846,Z 1021.339,A -85,B 0,C 180,E1 27601.928,E2 27601.928} C_VEL
LIN {X 0,Y 586.171,Z 1001.028,A -85,B 0,C 180,E1 27600.576,E2 27600.576} C_VEL
LIN {X 0,Y 586.595,Z 979.656,A -85,B 0,C 180,E1 27599.359,E2 27599.359} C_VEL
LIN {X 0,Y 586.875,Z 959.123,A -85,B 0,C 180,E1 27598.382,E2 27598.382} C_VEL
LIN {X 0,Y 587.251,Z 935.777,A -85,B 0,C 180,E1 27597.476,E2 27597.476} C_VEL
LIN {X 0,Y 587.467,Z 915.117,A -85,B 0,C 180,E1 27596.848,E2 27596.848} C_VEL
LIN {X 0,Y 587.712,Z 891.102,A -85,B 0,C 180,E1 27596.315,E2 27596.315} C_VEL
LIN {X 0,Y 588.402,Z 678.324,A -85,B 0,C 180,E1 27593.217,E2 27593.217} C_VEL
LIN {X 0,Y 588.697,Z 547.462,A -85,B 0,C 180,E1 27591.26,E2 27591.26} C_VEL
LIN {X 0,Y 587.75,Z 542.47,A -85,B 0,C 180,E1 27591.085,E2 27591.085} C_VEL
LIN {X 0,Y 587.972,Z 519.466,A -85,B 0,C 180,E1 27589.475,E2 27589.475} C_VEL
LIN {X 0,Y 584.101,Z 510.691,A -85,B 0,C 180,E1 27588.511,E2 27588.511} C_VEL
LIN {X 0,Y 584.048,Z 510.299,A -85,B 0,C 180,E1 27588.427,E2 27588.427} C_VEL
LIN {X 0,Y 584.055,Z 510.288,A -85,B 0,C 180,E1 27585.132,E2 27585.132} C_VEL
LIN {X 0,Y 584.055,Z 510.292,A -85,B 0,C 180,E1 27582.15,E2 27582.15} C_VEL
LIN {X 0,Y 584.06,Z 510.29,A -85,B 0,C 180,E1 27578.796,E2 27578.796} C_VEL
LIN {X 0,Y 584.076,Z 510.294,A -85,B 0,C 180,E1 27575.714,E2 27575.714} C_VEL
LIN {X 0,Y 584.062,Z 510.288,A -85,B 0,C 180,E1 27572.4,E2 27572.4} C_VEL
LIN {X 0,Y 584.099,Z 510.286,A -85,B 0,C 180,E1 27569.188,E2 27569.188} C_VEL
LIN {X 0,Y 584.064,Z 510.287,A -85,B 0,C 180,E1 27565.992,E2 27565.992} C_VEL
LIN {X 0,Y 584.092,Z 510.289,A -85,B 0,C 180,E1 27562.76,E2 27562.76} C_VEL
LIN {X 0,Y 584.067,Z 510.287,A -85,B 0,C 180,E1 27559.604,E2 27559.604} C_VEL
LIN {X 0,Y 584.087,Z 510.288,A -85,B 0,C 180,E1 27556.406,E2 27556.406} C_VEL
LIN {X 0,Y 584.073,Z 510.288,A -85,B 0,C 180,E1 27553.261,E2 27553.261} C_VEL
LIN {X 0,Y 584.082,Z 510.286,A -85,B 0,C 180,E1 27550.056,E2 27550.056} C_VEL
LIN {X 0,Y 584.079,Z 510.289,A -85,B 0,C 180,E1 27546.838,E2 27546.838} C_VEL
LIN {X 0,Y 584.079,Z 510.287,A -85,B 0,C 180,E1 27543.604,E2 27543.604} C_VEL
LIN {X 0,Y 584.086,Z 510.29,A -85,B 0,C 180,E1 27540.392,E2 27540.392} C_VEL
LIN {X 0,Y 584.077,Z 510.286,A -85,B 0,C 180,E1 27537.154,E2 27537.154} C_VEL
LIN {X 0,Y 584.093,Z 510.294,A -85,B 0,C 180,E1 27533.809,E2 27533.809} C_VEL
LIN {X 0,Y 584.095,Z 510.281,A -85,B 0,C 180,E1 27530.442,E2 27530.442} C_VEL
LIN {X 0,Y 584.064,Z 510.291,A -85,B 0,C 180,E1 27527.141,E2 27527.141} C_VEL
LIN {X 0,Y 584.065,Z 510.287,A -85,B 0,C 180,E1 27526.714,E2 27526.714} C_VEL
LIN {X 0,Y 583.111,Z 510.411,A -85,B 0,C 180,E1 27525.958,E2 27525.958} C_VEL
LIN {X 0,Y 576.614,Z 511.221,A -85,B 0,C 180,E1 27523.783,E2 27523.783} C_VEL
LIN {X 0,Y 576.143,Z 511.272,A -85,B 0,C 180,E1 27523.285,E2 27523.285} C_VEL
LIN {X 0,Y 576.148,Z 511.274,A -85,B 0,C 180,E1 27520.009,E2 27520.009} C_VEL
LIN {X 0,Y 576.115,Z 511.271,A -85,B 0,C 180,E1 27516.69,E2 27516.69} C_VEL
LIN {X 0,Y 576.158,Z 511.276,A -85,B 0,C 180,E1 27513.513,E2 27513.513} C_VEL
LIN {X 0,Y 576.105,Z 511.275,A -85,B 0,C 180,E1 27510.354,E2 27510.354} C_VEL
LIN {X 0,Y 576.156,Z 511.278,A -85,B 0,C 180,E1 27507.218,E2 27507.218} C_VEL
LIN {X 0,Y 576.095,Z 511.281,A -85,B 0,C 180,E1 27503.978,E2 27503.978} C_VEL
LIN {X 0,Y 576.156,Z 511.275,A -85,B 0,C 180,E1 27500.825,E2 27500.825} C_VEL
LIN {X 0,Y 576.085,Z 511.283,A -85,B 0,C 180,E1 27497.669,E2 27497.669} C_VEL
LIN {X 0,Y 576.136,Z 511.283,A -85,B 0,C 180,E1 27494.64,E2 27494.64} C_VEL
LIN {X 0,Y 576.076,Z 511.287,A -85,B 0,C 180,E1 27491.398,E2 27491.398} C_VEL
LIN {X 0,Y 576.132,Z 511.334,A -85,B 0,C 180,E1 27489.933,E2 27489.933} C_VEL
LIN {X 0,Y 577.02,Z 514.144,A -85,B 0,C 180,E1 27489.684,E2 27489.684} C_VEL
LIN {X 0,Y 582.559,Z 523.121,A -85,B 0,C 180,E1 27489.093,E2 27489.093} C_VEL
LIN {X 0,Y 581.775,Z 696.864,A -85,B 0,C 180,E1 27486.494,E2 27486.494} C_VEL
LIN {X 0,Y 581.04,Z 861.725,A -85,B 0,C 180,E1 27484.069,E2 27484.069} C_VEL
LIN {X 0,Y 580.712,Z 885.591,A -85,B 0,C 180,E1 27483.53,E2 27483.53} C_VEL
LIN {X 0,Y 580.415,Z 906.916,A -85,B 0,C 180,E1 27482.872,E2 27482.872} C_VEL
LIN {X 0,Y 579.923,Z 929.588,A -85,B 0,C 180,E1 27481.976,E2 27481.976} C_VEL
LIN {X 0,Y 579.525,Z 951.015,A -85,B 0,C 180,E1 27480.941,E2 27480.941} C_VEL
LIN {X 0,Y 578.958,Z 972.398,A -85,B 0,C 180,E1 27479.694,E2 27479.694} C_VEL
LIN {X 0,Y 578.475,Z 993.285,A -85,B 0,C 180,E1 27478.268,E2 27478.268} C_VEL
LIN {X 0,Y 577.997,Z 1011.885,A -85,B 0,C 180,E1 27476.796,E2 27476.796} C_VEL
LIN {X 0,Y 577.533,Z 1030.552,A -85,B 0,C 180,E1 27475.098,E2 27475.098} C_VEL
LIN {X 0,Y 577.165,Z 1047.489,A -85,B 0,C 180,E1 27473.342,E2 27473.342} C_VEL
LIN {X 0,Y 576.809,Z 1063.333,A -85,B 0,C 180,E1 27471.454,E2 27471.454} C_VEL
LIN {X 0,Y 576.52,Z 1078.642,A -85,B 0,C 180,E1 27469.359,E2 27469.359} C_VEL
LIN {X 0,Y 576.331,Z 1091.37,A -85,B 0,C 180,E1 27467.362,E2 27467.362} C_VEL
LIN {X 0,Y 576.153,Z 1102.944,A -85,B 0,C 180,E1 27465.229,E2 27465.229} C_VEL
LIN {X 0,Y 576.038,Z 1113.107,A -85,B 0,C 180,E1 27463.041,E2 27463.041} C_VEL
LIN {X 0,Y 575.97,Z 1121.247,A -85,B 0,C 180,E1 27460.908,E2 27460.908} C_VEL
LIN {X 0,Y 575.944,Z 1128.18,A -85,B 0,C 180,E1 27458.687,E2 27458.687} C_VEL
LIN {X 0,Y 575.912,Z 1133.16,A -85,B 0,C 180,E1 27456.58,E2 27456.58} C_VEL
LIN {X 0,Y 575.914,Z 1137.112,A -85,B 0,C 180,E1 27454.282,E2 27454.282} C_VEL
LIN {X 0,Y 575.914,Z 1139.226,A -85,B 0,C 180,E1 27452.09,E2 27452.09} C_VEL
LIN {X 0,Y 575.903,Z 1139.972,A -85,B 0,C 180,E1 27449.801,E2 27449.801} C_VEL
LIN {X 0,Y 575.916,Z 1139.152,A -85,B 0,C 180,E1 27447.712,E2 27447.712} C_VEL
LIN {X 0,Y 575.902,Z 1136.826,A -85,B 0,C 180,E1 27445.419,E2 27445.419} C_VEL
LIN {X 0,Y 575.901,Z 1132.934,A -85,B 0,C 180,E1 27443.22,E2 27443.22} C_VEL
LIN {X 0,Y 575.947,Z 1127.611,A -85,B 0,C 180,E1 27441.011,E2 27441.011} C_VEL
LIN {X 0,Y 575.965,Z 1120.853,A -85,B 0,C 180,E1 27438.89,E2 27438.89} C_VEL
LIN {X 0,Y 576.039,Z 1112.649,A -85,B 0,C 180,E1 27436.755,E2 27436.755} C_VEL
LIN {X 0,Y 576.151,Z 1102.544,A -85,B 0,C 180,E1 27434.602,E2 27434.602} C_VEL
LIN {X 0,Y 576.336,Z 1090.65,A -85,B 0,C 180,E1 27432.43,E2 27432.43} C_VEL
LIN {X 0,Y 576.539,Z 1077.927,A -85,B 0,C 180,E1 27430.445,E2 27430.445} C_VEL
LIN {X 0,Y 576.828,Z 1062.351,A -85,B 0,C 180,E1 27428.333,E2 27428.333} C_VEL
LIN {X 0,Y 577.19,Z 1046.591,A -85,B 0,C 180,E1 27426.466,E2 27426.466} C_VEL
LIN {X 0,Y 577.577,Z 1029.252,A -85,B 0,C 180,E1 27424.685,E2 27424.685} C_VEL
LIN {X 0,Y 578.035,Z 1009.797,A -85,B 0,C 180,E1 27422.94,E2 27422.94} C_VEL
LIN {X 0,Y 578.56,Z 990.795,A -85,B 0,C 180,E1 27421.455,E2 27421.455} C_VEL
LIN {X 0,Y 579.011,Z 970.506,A -85,B 0,C 180,E1 27420.097,E2 27420.097} C_VEL
LIN {X 0,Y 579.554,Z 948.448,A -85,B 0,C 180,E1 27418.838,E2 27418.838} C_VEL
LIN {X 0,Y 579.968,Z 927.99,A -85,B 0,C 180,E1 27417.864,E2 27417.864} C_VEL
LIN {X 0,Y 580.433,Z 904.958,A -85,B 0,C 180,E1 27416.972,E2 27416.972} C_VEL
LIN {X 0,Y 580.731,Z 883.969,A -85,B 0,C 180,E1 27416.335,E2 27416.335} C_VEL
LIN {X 0,Y 581.047,Z 860.638,A -85,B 0,C 180,E1 27415.823,E2 27415.823} C_VEL
LIN {X 0,Y 581.996,Z 648.252,A -85,B 0,C 180,E1 27412.698,E2 27412.698} C_VEL
LIN {X 0,Y 582.401,Z 522.656,A -85,B 0,C 180,E1 27410.797,E2 27410.797} C_VEL
LIN {X 0,Y 576.475,Z 512.889,A -85,B 0,C 180,E1 27410.129,E2 27410.129} C_VEL
LIN {X 0,Y 576.13,Z 511.286,A -85,B 0,C 180,E1 27409.938,E2 27409.938} C_VEL
LIN {X 0,Y 576.073,Z 511.287,A -85,B 0,C 180,E1 27406.8,E2 27406.8} C_VEL
LIN {X 0,Y 576.105,Z 511.286,A -85,B 0,C 180,E1 27403.925,E2 27403.925} C_VEL
LIN {X 0,Y 576.086,Z 511.282,A -85,B 0,C 180,E1 27400.606,E2 27400.606} C_VEL
LIN {X 0,Y 576.11,Z 511.28,A -85,B 0,C 180,E1 27397.683,E2 27397.683} C_VEL
LIN {X 0,Y 576.097,Z 511.274,A -85,B 0,C 180,E1 27394.337,E2 27394.337} C_VEL
LIN {X 0,Y 576.121,Z 511.284,A -85,B 0,C 180,E1 27391.365,E2 27391.365} C_VEL
LIN {X 0,Y 576.107,Z 511.277,A -85,B 0,C 180,E1 27388.056,E2 27388.056} C_VEL
LIN {X 0,Y 576.143,Z 511.281,A -85,B 0,C 180,E1 27384.943,E2 27384.943} C_VEL
LIN {X 0,Y 576.113,Z 511.276,A -85,B 0,C 180,E1 27381.695,E2 27381.695} C_VEL
LIN {X 0,Y 576.16,Z 511.275,A -85,B 0,C 180,E1 27378.517,E2 27378.517} C_VEL
LIN {X 0,Y 576.117,Z 511.275,A -85,B 0,C 180,E1 27375.296,E2 27375.296} C_VEL
LIN {X 0,Y 576.157,Z 511.279,A -85,B 0,C 180,E1 27372.122,E2 27372.122} C_VEL
LIN {X 0,Y 576.123,Z 511.277,A -85,B 0,C 180,E1 27368.886,E2 27368.886} C_VEL
LIN {X 0,Y 576.151,Z 511.276,A -85,B 0,C 180,E1 27365.677,E2 27365.677} C_VEL
LIN {X 0,Y 576.13,Z 511.279,A -85,B 0,C 180,E1 27362.487,E2 27362.487} C_VEL
LIN {X 0,Y 576.15,Z 511.275,A -85,B 0,C 180,E1 27359.205,E2 27359.205} C_VEL
LIN {X 0,Y 576.147,Z 511.28,A -85,B 0,C 180,E1 27355.92,E2 27355.92} C_VEL
LIN {X 0,Y 576.155,Z 511.273,A -85,B 0,C 180,E1 27352.522,E2 27352.522} C_VEL
LIN {X 0,Y 576.144,Z 511.271,A -85,B 0,C 180,E1 27349.191,E2 27349.191} C_VEL
LIN {X 0,Y 576.149,Z 511.275,A -85,B 0,C 180,E1 27345.939,E2 27345.939} C_VEL
LIN {X 0,Y 576.131,Z 511.27,A -85,B 0,C 180,E1 27342.737,E2 27342.737} C_VEL
LIN {X 0,Y 576.151,Z 511.277,A -85,B 0,C 180,E1 27339.479,E2 27339.479} C_VEL
LIN {X 0,Y 576.124,Z 511.272,A -85,B 0,C 180,E1 27336.366,E2 27336.366} C_VEL
LIN {X 0,Y 576.153,Z 511.28,A -85,B 0,C 180,E1 27333.126,E2 27333.126} C_VEL
LIN {X 0,Y 576.116,Z 511.277,A -85,B 0,C 180,E1 27330,E2 27330} C_VEL
LIN {X 0,Y 576.159,Z 511.278,A -85,B 0,C 180,E1 27326.744,E2 27326.744} C_VEL
LIN {X 0,Y 576.111,Z 511.28,A -85,B 0,C 180,E1 27323.591,E2 27323.591} C_VEL
LIN {X 0,Y 576.153,Z 511.281,A -85,B 0,C 180,E1 27320.311,E2 27320.311} C_VEL
LIN {X 0,Y 576.105,Z 511.279,A -85,B 0,C 180,E1 27317.234,E2 27317.234} C_VEL
LIN {X 0,Y 576.138,Z 511.285,A -85,B 0,C 180,E1 27313.929,E2 27313.929} C_VEL
LIN {X 0,Y 576.174,Z 511.399,A -85,B 0,C 180,E1 27312.137,E2 27312.137} C_VEL
LIN {X 0,Y 577.573,Z 514.973,A -85,B 0,C 180,E1 27311.745,E2 27311.745} C_VEL
LIN {X 0,Y 581.393,Z 523.232,A -85,B 0,C 180,E1 27310.807,E2 27310.807} C_VEL
LIN {X 0,Y 581.223,Z 543.465,A -85,B 0,C 180,E1 27309.396,E2 27309.396} C_VEL
LIN {X 0,Y 582.603,Z 551.122,A -85,B 0,C 180,E1 27309.165,E2 27309.165} C_VEL
LIN {X 0,Y 581.764,Z 730.715,A -85,B 0,C 180,E1 27306.482,E2 27306.482} C_VEL
LIN {X 0,Y 581.041,Z 891.668,A -85,B 0,C 180,E1 27304.114,E2 27304.114} C_VEL
LIN {X 0,Y 580.714,Z 915.474,A -85,B 0,C 180,E1 27303.578,E2 27303.578} C_VEL
LIN {X 0,Y 580.418,Z 936.71,A -85,B 0,C 180,E1 27302.924,E2 27302.924} C_VEL
LIN {X 0,Y 579.953,Z 958.409,A -85,B 0,C 180,E1 27302.073,E2 27302.073} C_VEL
LIN {X 0,Y 579.554,Z 978.549,A -85,B 0,C 180,E1 27301.111,E2 27301.111} C_VEL
LIN {X 0,Y 579.023,Z 1000.149,A -85,B 0,C 180,E1 27299.88,E2 27299.88} C_VEL
LIN {X 0,Y 578.575,Z 1020.19,A -85,B 0,C 180,E1 27298.544,E2 27298.544} C_VEL
LIN {X 0,Y 578.038,Z 1039.682,A -85,B 0,C 180,E1 27297.025,E2 27297.025} C_VEL
LIN {X 0,Y 577.575,Z 1059.352,A -85,B 0,C 180,E1 27295.26,E2 27295.26} C_VEL
LIN {X 0,Y 577.186,Z 1076.675,A -85,B 0,C 180,E1 27293.48,E2 27293.48} C_VEL
LIN {X 0,Y 576.818,Z 1092.844,A -85,B 0,C 180,E1 27291.56,E2 27291.56} C_VEL
LIN {X 0,Y 576.528,Z 1108.333,A -85,B 0,C 180,E1 27289.45,E2 27289.45} C_VEL
LIN {X 0,Y 576.327,Z 1121.644,A -85,B 0,C 180,E1 27287.361,E2 27287.361} C_VEL
LIN {X 0,Y 576.152,Z 1133.164,A -85,B 0,C 180,E1 27285.23,E2 27285.23} C_VEL
LIN {X 0,Y 576.037,Z 1143.289,A -85,B 0,C 180,E1 27283.041,E2 27283.041} C_VEL
LIN {X 0,Y 575.967,Z 1151.052,A -85,B 0,C 180,E1 27281.008,E2 27281.008} C_VEL
LIN {X 0,Y 575.943,Z 1158.04,A -85,B 0,C 180,E1 27278.787,E2 27278.787} C_VEL
LIN {X 0,Y 575.915,Z 1163.254,A -85,B 0,C 180,E1 27276.579,E2 27276.579} C_VEL
LIN {X 0,Y 575.914,Z 1167.164,A -85,B 0,C 180,E1 27274.281,E2 27274.281} C_VEL
LIN {X 0,Y 575.914,Z 1169.256,A -85,B 0,C 180,E1 27272.089,E2 27272.089} C_VEL
LIN {X 0,Y 575.899,Z 1169.962,A -85,B 0,C 180,E1 27269.801,E2 27269.801} C_VEL
LIN {X 0,Y 575.916,Z 1169.122,A -85,B 0,C 180,E1 27267.711,E2 27267.711} C_VEL
LIN {X 0,Y 575.904,Z 1166.753,A -85,B 0,C 180,E1 27265.419,E2 27265.419} C_VEL
LIN {X 0,Y 575.903,Z 1162.909,A -85,B 0,C 180,E1 27263.253,E2 27263.253} C_VEL
LIN {X 0,Y 575.947,Z 1157.475,A -85,B 0,C 180,E1 27261.011,E2 27261.011} C_VEL
LIN {X 0,Y 575.967,Z 1150.693,A -85,B 0,C 180,E1 27258.89,E2 27258.89} C_VEL
LIN {X 0,Y 576.037,Z 1142.455,A -85,B 0,C 180,E1 27256.754,E2 27256.754} C_VEL
LIN {X 0,Y 576.152,Z 1132.315,A -85,B 0,C 180,E1 27254.602,E2 27254.602} C_VEL
LIN {X 0,Y 576.338,Z 1120.374,A -85,B 0,C 180,E1 27252.43,E2 27252.43} C_VEL
LIN {X 0,Y 576.547,Z 1107.621,A -85,B 0,C 180,E1 27250.445,E2 27250.445} C_VEL
LIN {X 0,Y 576.818,Z 1092.84,A -85,B 0,C 180,E1 27248.439,E2 27248.439} C_VEL
LIN {X 0,Y 577.187,Z 1076.67,A -85,B 0,C 180,E1 27246.52,E2 27246.52} C_VEL
LIN {X 0,Y 577.574,Z 1059.347,A -85,B 0,C 180,E1 27244.74,E2 27244.74} C_VEL
LIN {X 0,Y 578.039,Z 1039.678,A -85,B 0,C 180,E1 27242.975,E2 27242.975} C_VEL
LIN {X 0,Y 578.575,Z 1020.181,A -85,B 0,C 180,E1 27241.456,E2 27241.456} C_VEL
LIN {X 0,Y 579.039,Z 999.691,A -85,B 0,C 180,E1 27240.092,E2 27240.092} C_VEL
LIN {X 0,Y 579.566,Z 977.423,A -85,B 0,C 180,E1 27238.831,E2 27238.831} C_VEL
LIN {X 0,Y 580,Z 956.987,A -85,B 0,C 180,E1 27237.865,E2 27237.865} C_VEL
LIN {X 0,Y 580.441,Z 934.165,A -85,B 0,C 180,E1 27236.991,E2 27236.991} C_VEL
LIN {X 0,Y 580.75,Z 913.269,A -85,B 0,C 180,E1 27236.361,E2 27236.361} C_VEL
LIN {X 0,Y 581.049,Z 890.16,A -85,B 0,C 180,E1 27235.86,E2 27235.86} C_VEL
LIN {X 0,Y 581.985,Z 679.723,A -85,B 0,C 180,E1 27232.764,E2 27232.764} C_VEL
LIN {X 0,Y 582.461,Z 549.314,A -85,B 0,C 180,E1 27230.795,E2 27230.795} C_VEL
LIN {X 0,Y 581.113,Z 542.855,A -85,B 0,C 180,E1 27230.582,E2 27230.582} C_VEL
LIN {X 0,Y 581.347,Z 523.084,A -85,B 0,C 180,E1 27229.178,E2 27229.178} C_VEL
LIN {X 0,Y 576.344,Z 512.281,A -85,B 0,C 180,E1 27227.945,E2 27227.945} C_VEL
LIN {X 0,Y 576.158,Z 511.283,A -85,B 0,C 180,E1 27227.817,E2 27227.817} C_VEL
LIN {X 0,Y 576.098,Z 511.279,A -85,B 0,C 180,E1 27224.635,E2 27224.635} C_VEL
LIN {X 0,Y 576.162,Z 511.279,A -85,B 0,C 180,E1 27221.436,E2 27221.436} C_VEL
LIN {X 0,Y 576.106,Z 511.282,A -85,B 0,C 180,E1 27218.286,E2 27218.286} C_VEL
LIN {X 0,Y 576.159,Z 511.271,A -85,B 0,C 180,E1 27215.058,E2 27215.058} C_VEL
LIN {X 0,Y 576.119,Z 511.28,A -85,B 0,C 180,E1 27211.843,E2 27211.843} C_VEL
LIN {X 0,Y 576.153,Z 511.27,A -85,B 0,C 180,E1 27208.505,E2 27208.505} C_VEL
LIN {X 0,Y 576.152,Z 511.279,A -85,B 0,C 180,E1 27205.161,E2 27205.161} C_VEL
LIN {X 0,Y 576.13,Z 511.274,A -85,B 0,C 180,E1 27201.8,E2 27201.8} C_VEL
LIN {X 0,Y 576.152,Z 511.271,A -85,B 0,C 180,E1 27198.621,E2 27198.621} C_VEL
LIN {X 0,Y 576.133,Z 511.275,A -85,B 0,C 180,E1 27195.398,E2 27195.398} C_VEL
LIN {X 0,Y 576.147,Z 511.272,A -85,B 0,C 180,E1 27192.223,E2 27192.223} C_VEL
LIN {X 0,Y 576.137,Z 511.273,A -85,B 0,C 180,E1 27188.986,E2 27188.986} C_VEL
LIN {X 0,Y 576.14,Z 511.275,A -85,B 0,C 180,E1 27185.777,E2 27185.777} C_VEL
LIN {X 0,Y 576.146,Z 511.28,A -85,B 0,C 180,E1 27182.486,E2 27182.486} C_VEL
LIN {X 0,Y 576.144,Z 511.274,A -85,B 0,C 180,E1 27179.204,E2 27179.204} C_VEL
LIN {X 0,Y 576.15,Z 511.281,A -85,B 0,C 180,E1 27175.82,E2 27175.82} C_VEL
LIN {X 0,Y 576.158,Z 511.274,A -85,B 0,C 180,E1 27172.521,E2 27172.521} C_VEL
LIN {X 0,Y 576.126,Z 511.272,A -85,B 0,C 180,E1 27169.197,E2 27169.197} C_VEL
LIN {X 0,Y 576.156,Z 511.277,A -85,B 0,C 180,E1 27165.953,E2 27165.953} C_VEL
LIN {X 0,Y 576.143,Z 511.272,A -85,B 0,C 180,E1 27163.285,E2 27163.285} C_VEL
LIN {X 0,Y 575.115,Z 511.395,A -85,B 0,C 180,E1 27162.52,E2 27162.52} C_VEL
LIN {X 0,Y 568.741,Z 512.197,A -85,B 0,C 180,E1 27160.369,E2 27160.369} C_VEL
LIN {X 0,Y 568.218,Z 512.264,A -85,B 0,C 180,E1 27159.81,E2 27159.81} C_VEL
LIN {X 0,Y 568.171,Z 512.257,A -85,B 0,C 180,E1 27156.565,E2 27156.565} C_VEL
LIN {X 0,Y 568.222,Z 512.267,A -85,B 0,C 180,E1 27153.339,E2 27153.339} C_VEL
LIN {X 0,Y 568.161,Z 512.262,A -85,B 0,C 180,E1 27150.181,E2 27150.181} C_VEL
LIN {X 0,Y 568.225,Z 512.27,A -85,B 0,C 180,E1 27146.942,E2 27146.942} C_VEL
LIN {X 0,Y 568.154,Z 512.27,A -85,B 0,C 180,E1 27143.75,E2 27143.75} C_VEL
LIN {X 0,Y 568.22,Z 512.261,A -85,B 0,C 180,E1 27140.563,E2 27140.563} C_VEL
LIN {X 0,Y 568.146,Z 512.272,A -85,B 0,C 180,E1 27137.485,E2 27137.485} C_VEL
LIN {X 0,Y 568.21,Z 512.265,A -85,B 0,C 180,E1 27134.26,E2 27134.26} C_VEL
LIN {X 0,Y 568.136,Z 512.277,A -85,B 0,C 180,E1 27131.129,E2 27131.129} C_VEL
LIN {X 0,Y 568.199,Z 512.416,A -85,B 0,C 180,E1 27130.519,E2 27130.519} C_VEL
LIN {X 0,Y 568.774,Z 514.409,A -85,B 0,C 180,E1 27130.373,E2 27130.373} C_VEL
LIN {X 0,Y 576.322,Z 526.244,A -85,B 0,C 180,E1 27129.55,E2 27129.55} C_VEL
LIN {X 0,Y 575.345,Z 696.534,A -85,B 0,C 180,E1 27126.975,E2 27126.975} C_VEL
LIN {X 0,Y 574.405,Z 861.769,A -85,B 0,C 180,E1 27124.517,E2 27124.517} C_VEL
LIN {X 0,Y 573.997,Z 885.655,A -85,B 0,C 180,E1 27123.974,E2 27123.974} C_VEL
LIN {X 0,Y 573.617,Z 907.414,A -85,B 0,C 180,E1 27123.295,E2 27123.295} C_VEL
LIN {X 0,Y 573.011,Z 929.979,A -85,B 0,C 180,E1 27122.391,E2 27122.391} C_VEL
LIN {X 0,Y 572.488,Z 951.351,A -85,B 0,C 180,E1 27121.346,E2 27121.346} C_VEL
LIN {X 0,Y 571.818,Z 972.123,A -85,B 0,C 180,E1 27120.122,E2 27120.122} C_VEL
LIN {X 0,Y 571.19,Z 993.291,A -85,B 0,C 180,E1 27118.662,E2 27118.662} C_VEL
LIN {X 0,Y 570.593,Z 1011.376,A -85,B 0,C 180,E1 27117.217,E2 27117.217} C_VEL
LIN {X 0,Y 570.029,Z 1030.006,A -85,B 0,C 180,E1 27115.507,E2 27115.507} C_VEL
LIN {X 0,Y 569.531,Z 1047.232,A -85,B 0,C 180,E1 27113.705,E2 27113.705} C_VEL
LIN {X 0,Y 569.071,Z 1063.339,A -85,B 0,C 180,E1 27111.761,E2 27111.761} C_VEL
LIN {X 0,Y 568.703,Z 1078.742,A -85,B 0,C 180,E1 27109.622,E2 27109.622} C_VEL
LIN {X 0,Y 568.436,Z 1091.988,A -85,B 0,C 180,E1 27107.505,E2 27107.505} C_VEL
LIN {X 0,Y 568.213,Z 1103.656,A -85,B 0,C 180,E1 27105.305,E2 27105.305} C_VEL
LIN {X 0,Y 568.067,Z 1113.929,A -85,B 0,C 180,E1 27103.02,E2 27103.02} C_VEL
LIN {X 0,Y 567.986,Z 1121.607,A -85,B 0,C 180,E1 27100.96,E2 27100.96} C_VEL
LIN {X 0,Y 567.947,Z 1128.692,A -85,B 0,C 180,E1 27098.606,E2 27098.606} C_VEL
LIN {X 0,Y 567.92,Z 1133.575,A -85,B 0,C 180,E1 27096.47,E2 27096.47} C_VEL
LIN {X 0,Y 567.917,Z 1137.452,A -85,B 0,C 180,E1 27094.039,E2 27094.039} C_VEL
LIN {X 0,Y 567.907,Z 1139.361,A -85,B 0,C 180,E1 27091.917,E2 27091.917} C_VEL
LIN {X 0,Y 567.885,Z 1139.905,A -85,B 0,C 180,E1 27089.496,E2 27089.496} C_VEL
LIN {X 0,Y 567.915,Z 1139.018,A -85,B 0,C 180,E1 27087.478,E2 27087.478} C_VEL
LIN {X 0,Y 567.906,Z 1136.347,A -85,B 0,C 180,E1 27085.051,E2 27085.051} C_VEL
LIN {X 0,Y 567.895,Z 1132.726,A -85,B 0,C 180,E1 27083.022,E2 27083.022} C_VEL
LIN {X 0,Y 567.944,Z 1127.003,A -85,B 0,C 180,E1 27080.679,E2 27080.679} C_VEL
LIN {X 0,Y 567.99,Z 1120.496,A -85,B 0,C 180,E1 27078.629,E2 27078.629} C_VEL
LIN {X 0,Y 568.081,Z 1111.738,A -85,B 0,C 180,E1 27076.359,E2 27076.359} C_VEL
LIN {X 0,Y 568.225,Z 1102.021,A -85,B 0,C 180,E1 27074.277,E2 27074.277} C_VEL
LIN {X 0,Y 568.45,Z 1090.009,A -85,B 0,C 180,E1 27072.073,E2 27072.073} C_VEL
LIN {X 0,Y 568.741,Z 1077.215,A -85,B 0,C 180,E1 27070.059,E2 27070.059} C_VEL
LIN {X 0,Y 569.099,Z 1062.347,A -85,B 0,C 180,E1 27068.024,E2 27068.024} C_VEL
LIN {X 0,Y 569.548,Z 1046.787,A -85,B 0,C 180,E1 27066.154,E2 27066.154} C_VEL
LIN {X 0,Y 570.056,Z 1029.245,A -85,B 0,C 180,E1 27064.327,E2 27064.327} C_VEL
LIN {X 0,Y 570.647,Z 1009.791,A -85,B 0,C 180,E1 27062.56,E2 27062.56} C_VEL
LIN {X 0,Y 571.277,Z 990.79,A -85,B 0,C 180,E1 27061.058,E2 27061.058} C_VEL
LIN {X 0,Y 571.866,Z 970.845,A -85,B 0,C 180,E1 27059.707,E2 27059.707} C_VEL
LIN {X 0,Y 572.523,Z 949.297,A -85,B 0,C 180,E1 27058.457,E2 27058.457} C_VEL
LIN {X 0,Y 573.06,Z 928.612,A -85,B 0,C 180,E1 27057.458,E2 27057.458} C_VEL
LIN {X 0,Y 573.637,Z 905.586,A -85,B 0,C 180,E1 27056.552,E2 27056.552} C_VEL
LIN {X 0,Y 574.019,Z 884.449,A -85,B 0,C 180,E1 27055.902,E2 27055.902} C_VEL
LIN {X 0,Y 574.413,Z 860.895,A -85,B 0,C 180,E1 27055.378,E2 27055.378} C_VEL
LIN {X 0,Y 575.608,Z 650.89,A -85,B 0,C 180,E1 27052.253,E2 27052.253} C_VEL
LIN {X 0,Y 576.154,Z 525.953,A -85,B 0,C 180,E1 27050.342,E2 27050.342} C_VEL
LIN {X 0,Y 570.27,Z 516.718,A -85,B 0,C 180,E1 27049.702,E2 27049.702} C_VEL
LIN {X 0,Y 568.431,Z 513.502,A -85,B 0,C 180,E1 27049.492,E2 27049.492} C_VEL
LIN {X 0,Y 568.164,Z 512.275,A -85,B 0,C 180,E1 27049.373,E2 27049.373} C_VEL
LIN {X 0,Y 568.136,Z 512.277,A -85,B 0,C 180,E1 27046.38,E2 27046.38} C_VEL
LIN {X 0,Y 568.177,Z 512.272,A -85,B 0,C 180,E1 27043.088,E2 27043.088} C_VEL
LIN {X 0,Y 568.146,Z 512.272,A -85,B 0,C 180,E1 27040.099,E2 27040.099} C_VEL
LIN {X 0,Y 568.187,Z 512.269,A -85,B 0,C 180,E1 27036.805,E2 27036.805} C_VEL
LIN {X 0,Y 568.157,Z 512.263,A -85,B 0,C 180,E1 27033.787,E2 27033.787} C_VEL
LIN {X 0,Y 568.203,Z 512.261,A -85,B 0,C 180,E1 27030.567,E2 27030.567} C_VEL
LIN {X 0,Y 568.167,Z 512.268,A -85,B 0,C 180,E1 27027.456,E2 27027.456} C_VEL
LIN {X 0,Y 568.192,Z 512.256,A -85,B 0,C 180,E1 27024.095,E2 27024.095} C_VEL
LIN {X 0,Y 568.192,Z 512.269,A -85,B 0,C 180,E1 27020.93,E2 27020.93} C_VEL
LIN {X 0,Y 568.185,Z 512.256,A -85,B 0,C 180,E1 27017.619,E2 27017.619} C_VEL
LIN {X 0,Y 568.221,Z 512.27,A -85,B 0,C 180,E1 27014.366,E2 27014.366} C_VEL
LIN {X 0,Y 568.183,Z 512.265,A -85,B 0,C 180,E1 27011.059,E2 27011.059} C_VEL
LIN {X 0,Y 568.214,Z 512.267,A -85,B 0,C 180,E1 27007.787,E2 27007.787} C_VEL
LIN {X 0,Y 568.19,Z 512.266,A -85,B 0,C 180,E1 27004.542,E2 27004.542} C_VEL
LIN {X 0,Y 568.217,Z 512.26,A -85,B 0,C 180,E1 27001.21,E2 27001.21} C_VEL
LIN {X 0,Y 568.217,Z 512.269,A -85,B 0,C 180,E1 26997.782,E2 26997.782} C_VEL
LIN {X 0,Y 568.206,Z 512.263,A -85,B 0,C 180,E1 26994.446,E2 26994.446} C_VEL
LIN {X 0,Y 568.205,Z 512.266,A -85,B 0,C 180,E1 26991.194,E2 26991.194} C_VEL
LIN {X 0,Y 568.205,Z 512.255,A -85,B 0,C 180,E1 26987.913,E2 26987.913} C_VEL
LIN {X 0,Y 568.196,Z 512.265,A -85,B 0,C 180,E1 26984.695,E2 26984.695} C_VEL
LIN {X 0,Y 568.212,Z 512.257,A -85,B 0,C 180,E1 26981.428,E2 26981.428} C_VEL
LIN {X 0,Y 568.193,Z 512.264,A -85,B 0,C 180,E1 26978.205,E2 26978.205} C_VEL
LIN {X 0,Y 568.212,Z 512.268,A -85,B 0,C 180,E1 26974.797,E2 26974.797} C_VEL
LIN {X 0,Y 568.222,Z 512.259,A -85,B 0,C 180,E1 26971.405,E2 26971.405} C_VEL
LIN {X 0,Y 568.181,Z 512.269,A -85,B 0,C 180,E1 26968.135,E2 26968.135} C_VEL
LIN {X 0,Y 568.22,Z 512.261,A -85,B 0,C 180,E1 26964.873,E2 26964.873} C_VEL
LIN {X 0,Y 568.168,Z 512.264,A -85,B 0,C 180,E1 26961.709,E2 26961.709} C_VEL
LIN {X 0,Y 568.223,Z 512.265,A -85,B 0,C 180,E1 26958.556,E2 26958.556} C_VEL
LIN {X 0,Y 568.161,Z 512.271,A -85,B 0,C 180,E1 26955.314,E2 26955.314} C_VEL
LIN {X 0,Y 568.204,Z 512.489,A -85,B 0,C 180,E1 26952.784,E2 26952.784} C_VEL
LIN {X 0,Y 569.265,Z 515.369,A -85,B 0,C 180,E1 26952.466,E2 26952.466} C_VEL
LIN {X 0,Y 574.793,Z 527.192,A -85,B 0,C 180,E1 26951.084,E2 26951.084} C_VEL
LIN {X 0,Y 574.645,Z 543.581,A -85,B 0,C 180,E1 26949.935,E2 26949.935} C_VEL
LIN {X 0,Y 576.385,Z 552.751,A -85,B 0,C 180,E1 26949.645,E2 26949.645} C_VEL
LIN {X 0,Y 575.319,Z 732.542,A -85,B 0,C 180,E1 26946.93,E2 26946.93} C_VEL
LIN {X 0,Y 574.407,Z 891.775,A -85,B 0,C 180,E1 26944.562,E2 26944.562} C_VEL
LIN {X 0,Y 573.996,Z 915.628,A -85,B 0,C 180,E1 26944.02,E2 26944.02} C_VEL
LIN {X 0,Y 573.615,Z 937.423,A -85,B 0,C 180,E1 26943.34,E2 26943.34} C_VEL
LIN {X 0,Y 573.021,Z 959.685,A -85,B 0,C 180,E1 26942.449,E2 26942.449} C_VEL
LIN {X 0,Y 572.503,Z 980.787,A -85,B 0,C 180,E1 26941.421,E2 26941.421} C_VEL
LIN {X 0,Y 571.826,Z 1001.934,A -85,B 0,C 180,E1 26940.179,E2 26940.179} C_VEL
LIN {X 0,Y 571.197,Z 1023.113,A -85,B 0,C 180,E1 26938.721,E2 26938.721} C_VEL
LIN {X 0,Y 570.595,Z 1041.249,A -85,B 0,C 180,E1 26937.273,E2 26937.273} C_VEL
LIN {X 0,Y 570.012,Z 1060.458,A -85,B 0,C 180,E1 26935.508,E2 26935.508} C_VEL
LIN {X 0,Y 569.516,Z 1077.617,A -85,B 0,C 180,E1 26933.706,E2 26933.706} C_VEL
LIN {X 0,Y 569.063,Z 1093.694,A -85,B 0,C 180,E1 26931.761,E2 26931.761} C_VEL
LIN {X 0,Y 568.714,Z 1108.335,A -85,B 0,C 180,E1 26929.728,E2 26929.728} C_VEL
LIN {X 0,Y 568.446,Z 1121.009,A -85,B 0,C 180,E1 26927.716,E2 26927.716} C_VEL
LIN {X 0,Y 568.22,Z 1132.318,A -85,B 0,C 180,E1 26925.618,E2 26925.618} C_VEL
LIN {X 0,Y 568.075,Z 1142.456,A -85,B 0,C 180,E1 26923.434,E2 26923.434} C_VEL
LIN {X 0,Y 567.988,Z 1150.696,A -85,B 0,C 180,E1 26921.268,E2 26921.268} C_VEL
LIN {X 0,Y 567.954,Z 1157.476,A -85,B 0,C 180,E1 26919.116,E2 26919.116} C_VEL
LIN {X 0,Y 567.899,Z 1162.841,A -85,B 0,C 180,E1 26916.876,E2 26916.876} C_VEL
LIN {X 0,Y 567.904,Z 1166.595,A -85,B 0,C 180,E1 26914.746,E2 26914.746} C_VEL
LIN {X 0,Y 567.915,Z 1169.055,A -85,B 0,C 180,E1 26912.421,E2 26912.421} C_VEL
LIN {X 0,Y 567.892,Z 1169.939,A -85,B 0,C 180,E1 26910.302,E2 26910.302} C_VEL
LIN {X 0,Y 567.91,Z 1169.323,A -85,B 0,C 180,E1 26907.982,E2 26907.982} C_VEL
LIN {X 0,Y 567.916,Z 1167.276,A -85,B 0,C 180,E1 26905.759,E2 26905.759} C_VEL
LIN {X 0,Y 567.919,Z 1163.46,A -85,B 0,C 180,E1 26903.429,E2 26903.429} C_VEL
LIN {X 0,Y 567.948,Z 1158.55,A -85,B 0,C 180,E1 26901.292,E2 26901.292} C_VEL
LIN {X 0,Y 567.984,Z 1151.763,A -85,B 0,C 180,E1 26899.04,E2 26899.04} C_VEL
LIN {X 0,Y 568.066,Z 1144.107,A -85,B 0,C 180,E1 26896.98,E2 26896.98} C_VEL
LIN {X 0,Y 568.211,Z 1133.61,A -85,B 0,C 180,E1 26894.641,E2 26894.641} C_VEL
LIN {X 0,Y 568.43,Z 1122.235,A -85,B 0,C 180,E1 26892.495,E2 26892.495} C_VEL
LIN {X 0,Y 568.694,Z 1109.041,A -85,B 0,C 180,E1 26890.378,E2 26890.378} C_VEL
LIN {X 0,Y 569.045,Z 1094.535,A -85,B 0,C 180,E1 26888.346,E2 26888.346} C_VEL
LIN {X 0,Y 569.45,Z 1079.474,A -85,B 0,C 180,E1 26886.511,E2 26886.511} C_VEL
LIN {X 0,Y 569.95,Z 1062.112,A -85,B 0,C 180,E1 26884.656,E2 26884.656} C_VEL
LIN {X 0,Y 570.536,Z 1043.888,A -85,B 0,C 180,E1 26882.949,E2 26882.949} C_VEL
LIN {X 0,Y 571.141,Z 1024.604,A -85,B 0,C 180,E1 26881.393,E2 26881.393} C_VEL
LIN {X 0,Y 571.765,Z 1003.706,A -85,B 0,C 180,E1 26879.933,E2 26879.933} C_VEL
LIN {X 0,Y 572.4,Z 983.823,A -85,B 0,C 180,E1 26878.748,E2 26878.748} C_VEL
LIN {X 0,Y 572.972,Z 961.419,A -85,B 0,C 180,E1 26877.628,E2 26877.628} C_VEL
LIN {X 0,Y 573.582,Z 939.354,A -85,B 0,C 180,E1 26876.727,E2 26876.727} C_VEL
LIN {X 0,Y 573.982,Z 916.824,A -85,B 0,C 180,E1 26876.013,E2 26876.013} C_VEL
LIN {X 0,Y 574.393,Z 893.886,A -85,B 0,C 180,E1 26875.474,E2 26875.474} C_VEL
LIN {X 0,Y 574.752,Z 837.777,A -85,B 0,C 180,E1 26874.623,E2 26874.623} C_VEL
LIN {X 0,Y 575.981,Z 624.537,A -85,B 0,C 180,E1 26871.452,E2 26871.452} C_VEL
LIN {X 0,Y 576.217,Z 550.908,A -85,B 0,C 180,E1 26870.312,E2 26870.312} C_VEL
LIN {X 0,Y 574.511,Z 542.47,A -85,B 0,C 180,E1 26870.011,E2 26870.011} C_VEL
LIN {X 0,Y 574.655,Z 526.925,A -85,B 0,C 180,E1 26868.884,E2 26868.884} C_VEL
LIN {X 0,Y 569.735,Z 516.062,A -85,B 0,C 180,E1 26867.63,E2 26867.63} C_VEL
LIN {X 0,Y 568.323,Z 513.082,A -85,B 0,C 180,E1 26867.272,E2 26867.272} C_VEL
LIN {X 0,Y 568.173,Z 512.274,A -85,B 0,C 180,E1 26867.181,E2 26867.181} C_VEL
LIN {X 0,Y 568.186,Z 512.27,A -85,B 0,C 180,E1 26864.112,E2 26864.112} C_VEL
LIN {X 0,Y 568.173,Z 512.27,A -85,B 0,C 180,E1 26860.758,E2 26860.758} C_VEL
LIN {X 0,Y 568.211,Z 512.271,A -85,B 0,C 180,E1 26857.633,E2 26857.633} C_VEL
LIN {X 0,Y 568.176,Z 512.261,A -85,B 0,C 180,E1 26854.377,E2 26854.377} C_VEL
LIN {X 0,Y 568.219,Z 512.266,A -85,B 0,C 180,E1 26851.153,E2 26851.153} C_VEL
LIN {X 0,Y 568.179,Z 512.263,A -85,B 0,C 180,E1 26847.91,E2 26847.91} C_VEL
LIN {X 0,Y 568.214,Z 512.258,A -85,B 0,C 180,E1 26844.758,E2 26844.758} C_VEL
LIN {X 0,Y 568.189,Z 512.265,A -85,B 0,C 180,E1 26841.47,E2 26841.47} C_VEL
LIN {X 0,Y 568.216,Z 512.252,A -85,B 0,C 180,E1 26838.147,E2 26838.147} C_VEL
LIN {X 0,Y 568.211,Z 512.269,A -85,B 0,C 180,E1 26834.782,E2 26834.782} C_VEL
LIN {X 0,Y 568.204,Z 512.256,A -85,B 0,C 180,E1 26831.366,E2 26831.366} C_VEL
LIN {X 0,Y 568.206,Z 512.269,A -85,B 0,C 180,E1 26828.092,E2 26828.092} C_VEL
LIN {X 0,Y 568.203,Z 512.263,A -85,B 0,C 180,E1 26824.845,E2 26824.845} C_VEL
LIN {X 0,Y 568.199,Z 512.266,A -85,B 0,C 180,E1 26821.613,E2 26821.613} C_VEL
LIN {X 0,Y 568.209,Z 512.267,A -85,B 0,C 180,E1 26818.386,E2 26818.386} C_VEL
LIN {X 0,Y 568.194,Z 512.263,A -85,B 0,C 180,E1 26815.154,E2 26815.154} C_VEL
LIN {X 0,Y 568.218,Z 512.269,A -85,B 0,C 180,E1 26811.805,E2 26811.805} C_VEL
LIN {X 0,Y 568.212,Z 512.254,A -85,B 0,C 180,E1 26808.428,E2 26808.428} C_VEL
LIN {X 0,Y 568.187,Z 512.268,A -85,B 0,C 180,E1 26805.112,E2 26805.112} C_VEL
LIN {X 0,Y 568.219,Z 512.253,A -85,B 0,C 180,E1 26801.844,E2 26801.844} C_VEL
LIN {X 0,Y 568.218,Z 512.264,A -85,B 0,C 180,E1 26799.81,E2 26799.81} C_VEL
LIN {X 0,Y 567.221,Z 512.393,A -85,B 0,C 180,E1 26799.033,E2 26799.033} C_VEL
LIN {X 0,Y 560.753,Z 513.184,A -85,B 0,C 180,E1 26796.853,E2 26796.853} C_VEL
LIN {X 0,Y 560.232,Z 513.242,A -85,B 0,C 180,E1 26796.285,E2 26796.285} C_VEL
LIN {X 0,Y 560.269,Z 513.259,A -85,B 0,C 180,E1 26792.93,E2 26792.93} C_VEL
LIN {X 0,Y 560.234,Z 513.248,A -85,B 0,C 180,E1 26789.747,E2 26789.747} C_VEL
LIN {X 0,Y 560.229,Z 513.253,A -85,B 0,C 180,E1 26786.286,E2 26786.286} C_VEL
LIN {X 0,Y 560.255,Z 513.257,A -85,B 0,C 180,E1 26783.156,E2 26783.156} C_VEL
LIN {X 0,Y 560.215,Z 513.261,A -85,B 0,C 180,E1 26779.886,E2 26779.886} C_VEL
LIN {X 0,Y 560.243,Z 513.26,A -85,B 0,C 180,E1 26776.879,E2 26776.879} C_VEL
LIN {X 0,Y 560.204,Z 513.251,A -85,B 0,C 180,E1 26773.561,E2 26773.561} C_VEL
LIN {X 0,Y 560.225,Z 513.462,A -85,B 0,C 180,E1 26771.138,E2 26771.138} C_VEL
LIN {X 0,Y 561.485,Z 516.714,A -85,B 0,C 180,E1 26770.972,E2 26770.972} C_VEL
LIN {X 0,Y 563.631,Z 519.392,A -85,B 0,C 180,E1 26770.738,E2 26770.738} C_VEL
LIN {X 0,Y 570.132,Z 529.882,A -85,B 0,C 180,E1 26770.007,E2 26770.007} C_VEL
LIN {X 0,Y 568.904,Z 705.324,A -85,B 0,C 180,E1 26767.329,E2 26767.329} C_VEL
LIN {X 0,Y 567.807,Z 861.919,A -85,B 0,C 180,E1 26764.975,E2 26764.975} C_VEL
LIN {X 0,Y 567.326,Z 885.631,A -85,B 0,C 180,E1 26764.431,E2 26764.431} C_VEL
LIN {X 0,Y 566.854,Z 907.526,A -85,B 0,C 180,E1 26763.743,E2 26763.743} C_VEL
LIN {X 0,Y 566.152,Z 929.999,A -85,B 0,C 180,E1 26762.833,E2 26762.833} C_VEL
LIN {X 0,Y 565.499,Z 951.042,A -85,B 0,C 180,E1 26761.796,E2 26761.796} C_VEL
LIN {X 0,Y 564.751,Z 971.16,A -85,B 0,C 180,E1 26760.604,E2 26760.604} C_VEL
LIN {X 0,Y 563.983,Z 991.829,A -85,B 0,C 180,E1 26759.179,E2 26759.179} C_VEL
LIN {X 0,Y 563.269,Z 1010.063,A -85,B 0,C 180,E1 26757.716,E2 26757.716} C_VEL
LIN {X 0,Y 562.541,Z 1029.489,A -85,B 0,C 180,E1 26755.925,E2 26755.925} C_VEL
LIN {X 0,Y 561.923,Z 1046.754,A -85,B 0,C 180,E1 26754.104,E2 26754.104} C_VEL
LIN {X 0,Y 561.369,Z 1062.74,A -85,B 0,C 180,E1 26752.154,E2 26752.154} C_VEL
LIN {X 0,Y 560.911,Z 1078.04,A -85,B 0,C 180,E1 26750.014,E2 26750.014} C_VEL
LIN {X 0,Y 560.564,Z 1090.739,A -85,B 0,C 180,E1 26747.974,E2 26747.974} C_VEL
LIN {X 0,Y 560.3,Z 1102.098,A -85,B 0,C 180,E1 26745.845,E2 26745.845} C_VEL
LIN {X 0,Y 560.129,Z 1111.799,A -85,B 0,C 180,E1 26743.734,E2 26743.734} C_VEL
LIN {X 0,Y 560.02,Z 1120.561,A -85,B 0,C 180,E1 26741.425,E2 26741.425} C_VEL
LIN {X 0,Y 559.951,Z 1127.342,A -85,B 0,C 180,E1 26739.248,E2 26739.248} C_VEL
LIN {X 0,Y 559.897,Z 1132.75,A -85,B 0,C 180,E1 26736.975,E2 26736.975} C_VEL
LIN {X 0,Y 559.91,Z 1136.501,A -85,B 0,C 180,E1 26734.83,E2 26734.83} C_VEL
LIN {X 0,Y 559.913,Z 1139.025,A -85,B 0,C 180,E1 26732.457,E2 26732.457} C_VEL
LIN {X 0,Y 559.894,Z 1139.929,A -85,B 0,C 180,E1 26730.307,E2 26730.307} C_VEL
LIN {X 0,Y 559.911,Z 1139.353,A -85,B 0,C 180,E1 26727.953,E2 26727.953} C_VEL
LIN {X 0,Y 559.916,Z 1137.44,A -85,B 0,C 180,E1 26725.802,E2 26725.802} C_VEL
LIN {X 0,Y 559.917,Z 1133.551,A -85,B 0,C 180,E1 26723.335,E2 26723.335} C_VEL
LIN {X 0,Y 559.951,Z 1128.917,A -85,B 0,C 180,E1 26721.27,E2 26721.27} C_VEL
LIN {X 0,Y 559.998,Z 1121.919,A -85,B 0,C 180,E1 26718.882,E2 26718.882} C_VEL
LIN {X 0,Y 560.098,Z 1114.285,A -85,B 0,C 180,E1 26716.791,E2 26716.791} C_VEL
LIN {X 0,Y 560.274,Z 1104.103,A -85,B 0,C 180,E1 26714.473,E2 26714.473} C_VEL
LIN {X 0,Y 560.527,Z 1093.063,A -85,B 0,C 180,E1 26712.348,E2 26712.348} C_VEL
LIN {X 0,Y 560.855,Z 1080.048,A -85,B 0,C 180,E1 26710.201,E2 26710.201} C_VEL
LIN {X 0,Y 561.284,Z 1065.714,A -85,B 0,C 180,E1 26708.14,E2 26708.14} C_VEL
LIN {X 0,Y 561.8,Z 1049.854,A -85,B 0,C 180,E1 26706.172,E2 26706.172} C_VEL
LIN {X 0,Y 562.435,Z 1032.154,A -85,B 0,C 180,E1 26704.252,E2 26704.252} C_VEL
LIN {X 0,Y 563.096,Z 1014.819,A -85,B 0,C 180,E1 26702.601,E2 26702.601} C_VEL
LIN {X 0,Y 563.821,Z 995.908,A -85,B 0,C 180,E1 26701.045,E2 26701.045} C_VEL
LIN {X 0,Y 564.585,Z 975.288,A -85,B 0,C 180,E1 26699.569,E2 26699.569} C_VEL
LIN {X 0,Y 565.323,Z 955.592,A -85,B 0,C 180,E1 26698.372,E2 26698.372} C_VEL
LIN {X 0,Y 566.045,Z 933.273,A -85,B 0,C 180,E1 26697.225,E2 26697.225} C_VEL
LIN {X 0,Y 566.689,Z 912.607,A -85,B 0,C 180,E1 26696.357,E2 26696.357} C_VEL
LIN {X 0,Y 567.263,Z 889.419,A -85,B 0,C 180,E1 26695.586,E2 26695.586} C_VEL
LIN {X 0,Y 567.684,Z 868.037,A -85,B 0,C 180,E1 26695.054,E2 26695.054} C_VEL
LIN {X 0,Y 568.036,Z 836.706,A -85,B 0,C 180,E1 26694.537,E2 26694.537} C_VEL
LIN {X 0,Y 569.447,Z 630.342,A -85,B 0,C 180,E1 26691.449,E2 26691.449} C_VEL
LIN {X 0,Y 570.029,Z 529.402,A -85,B 0,C 180,E1 26689.886,E2 26689.886} C_VEL
LIN {X 0,Y 564.933,Z 521.627,A -85,B 0,C 180,E1 26689.323,E2 26689.323} C_VEL
LIN {X 0,Y 562.747,Z 518.188,A -85,B 0,C 180,E1 26689.075,E2 26689.075} C_VEL
LIN {X 0,Y 560.683,Z 515.203,A -85,B 0,C 180,E1 26688.842,E2 26688.842} C_VEL
LIN {X 0,Y 560.19,Z 513.268,A -85,B 0,C 180,E1 26688.742,E2 26688.742} C_VEL
LIN {X 0,Y 560.274,Z 513.262,A -85,B 0,C 180,E1 26685.548,E2 26685.548} C_VEL
LIN {X 0,Y 560.2,Z 513.263,A -85,B 0,C 180,E1 26682.361,E2 26682.361} C_VEL
LIN {X 0,Y 560.278,Z 513.248,A -85,B 0,C 180,E1 26679.179,E2 26679.179} C_VEL
LIN {X 0,Y 560.21,Z 513.26,A -85,B 0,C 180,E1 26676.049,E2 26676.049} C_VEL
LIN {X 0,Y 560.279,Z 513.258,A -85,B 0,C 180,E1 26672.803,E2 26672.803} C_VEL
LIN {X 0,Y 560.222,Z 513.253,A -85,B 0,C 180,E1 26669.629,E2 26669.629} C_VEL
LIN {X 0,Y 560.271,Z 513.255,A -85,B 0,C 180,E1 26666.38,E2 26666.38} C_VEL
LIN {X 0,Y 560.236,Z 513.247,A -85,B 0,C 180,E1 26663.201,E2 26663.201} C_VEL
LIN {X 0,Y 560.253,Z 513.254,A -85,B 0,C 180,E1 26659.821,E2 26659.821} C_VEL
LIN {X 0,Y 560.269,Z 513.245,A -85,B 0,C 180,E1 26656.591,E2 26656.591} C_VEL
LIN {X 0,Y 560.248,Z 513.255,A -85,B 0,C 180,E1 26653.31,E2 26653.31} C_VEL
LIN {X 0,Y 560.278,Z 513.258,A -85,B 0,C 180,E1 26650.072,E2 26650.072} C_VEL
LIN {X 0,Y 560.249,Z 513.256,A -85,B 0,C 180,E1 26646.765,E2 26646.765} C_VEL
LIN {X 0,Y 560.274,Z 513.255,A -85,B 0,C 180,E1 26643.479,E2 26643.479} C_VEL
LIN {X 0,Y 560.26,Z 513.255,A -85,B 0,C 180,E1 26640.205,E2 26640.205} C_VEL
LIN {X 0,Y 560.279,Z 513.25,A -85,B 0,C 180,E1 26636.829,E2 26636.829} C_VEL
LIN {X 0,Y 560.274,Z 513.259,A -85,B 0,C 180,E1 26633.442,E2 26633.442} C_VEL
LIN {X 0,Y 560.267,Z 513.25,A -85,B 0,C 180,E1 26630.099,E2 26630.099} C_VEL
LIN {X 0,Y 560.26,Z 513.255,A -85,B 0,C 180,E1 26626.795,E2 26626.795} C_VEL
LIN {X 0,Y 560.272,Z 513.256,A -85,B 0,C 180,E1 26623.516,E2 26623.516} C_VEL
LIN {X 0,Y 560.262,Z 513.253,A -85,B 0,C 180,E1 26620.18,E2 26620.18} C_VEL
LIN {X 0,Y 560.266,Z 513.247,A -85,B 0,C 180,E1 26616.772,E2 26616.772} C_VEL
LIN {X 0,Y 560.28,Z 513.254,A -85,B 0,C 180,E1 26613.389,E2 26613.389} C_VEL
LIN {X 0,Y 560.242,Z 513.255,A -85,B 0,C 180,E1 26610.137,E2 26610.137} C_VEL
LIN {X 0,Y 560.281,Z 513.254,A -85,B 0,C 180,E1 26606.902,E2 26606.902} C_VEL
LIN {X 0,Y 560.233,Z 513.259,A -85,B 0,C 180,E1 26603.664,E2 26603.664} C_VEL
LIN {X 0,Y 560.281,Z 513.254,A -85,B 0,C 180,E1 26600.425,E2 26600.425} C_VEL
LIN {X 0,Y 560.226,Z 513.257,A -85,B 0,C 180,E1 26597.297,E2 26597.297} C_VEL
LIN {X 0,Y 560.265,Z 513.262,A -85,B 0,C 180,E1 26593.965,E2 26593.965} C_VEL
LIN {X 0,Y 560.243,Z 513.413,A -85,B 0,C 180,E1 26593.469,E2 26593.469} C_VEL
LIN {X 0,Y 561.448,Z 516.629,A -85,B 0,C 180,E1 26593.101,E2 26593.101} C_VEL
LIN {X 0,Y 565.957,Z 526.158,A -85,B 0,C 180,E1 26591.947,E2 26591.947} C_VEL
LIN {X 0,Y 568.222,Z 531.125,A -85,B 0,C 180,E1 26591.369,E2 26591.369} C_VEL
LIN {X 0,Y 568.063,Z 543.521,A -85,B 0,C 180,E1 26590.494,E2 26590.494} C_VEL
LIN {X 0,Y 570.208,Z 554.48,A -85,B 0,C 180,E1 26590.133,E2 26590.133} C_VEL
LIN {X 0,Y 568.908,Z 734.727,A -85,B 0,C 180,E1 26587.383,E2 26587.383} C_VEL
LIN {X 0,Y 567.809,Z 891.883,A -85,B 0,C 180,E1 26585.02,E2 26585.02} C_VEL
LIN {X 0,Y 567.322,Z 915.757,A -85,B 0,C 180,E1 26584.473,E2 26584.473} C_VEL
LIN {X 0,Y 566.849,Z 937.742,A -85,B 0,C 180,E1 26583.78,E2 26583.78} C_VEL
LIN {X 0,Y 566.165,Z 959.689,A -85,B 0,C 180,E1 26582.892,E2 26582.892} C_VEL
LIN {X 0,Y 565.506,Z 980.789,A -85,B 0,C 180,E1 26581.855,E2 26581.855} C_VEL
LIN {X 0,Y 564.722,Z 1001.848,A -85,B 0,C 180,E1 26580.605,E2 26580.605} C_VEL
LIN {X 0,Y 563.96,Z 1022.406,A -85,B 0,C 180,E1 26579.18,E2 26579.18} C_VEL
LIN {X 0,Y 563.249,Z 1040.59,A -85,B 0,C 180,E1 26577.716,E2 26577.716} C_VEL
LIN {X 0,Y 562.523,Z 1059.964,A -85,B 0,C 180,E1 26575.923,E2 26575.923} C_VEL
LIN {X 0,Y 561.91,Z 1077.158,A -85,B 0,C 180,E1 26574.102,E2 26574.102} C_VEL
LIN {X 0,Y 561.36,Z 1093.097,A -85,B 0,C 180,E1 26572.152,E2 26572.152} C_VEL
LIN {X 0,Y 560.903,Z 1108.337,A -85,B 0,C 180,E1 26570.014,E2 26570.014} C_VEL
LIN {X 0,Y 560.561,Z 1121.007,A -85,B 0,C 180,E1 26567.973,E2 26567.973} C_VEL
LIN {X 0,Y 560.297,Z 1132.319,A -85,B 0,C 180,E1 26565.845,E2 26565.845} C_VEL
LIN {X 0,Y 560.127,Z 1141.996,A -85,B 0,C 180,E1 26563.734,E2 26563.734} C_VEL
LIN {X 0,Y 560.015,Z 1150.716,A -85,B 0,C 180,E1 26561.425,E2 26561.425} C_VEL
LIN {X 0,Y 559.955,Z 1157.475,A -85,B 0,C 180,E1 26559.248,E2 26559.248} C_VEL
LIN {X 0,Y 559.899,Z 1162.841,A -85,B 0,C 180,E1 26556.975,E2 26556.975} C_VEL
LIN {X 0,Y 559.906,Z 1166.595,A -85,B 0,C 180,E1 26554.814,E2 26554.814} C_VEL
LIN {X 0,Y 559.915,Z 1169.055,A -85,B 0,C 180,E1 26552.456,E2 26552.456} C_VEL
LIN {X 0,Y 559.892,Z 1169.939,A -85,B 0,C 180,E1 26550.307,E2 26550.307} C_VEL
LIN {X 0,Y 559.911,Z 1169.323,A -85,B 0,C 180,E1 26547.953,E2 26547.953} C_VEL
LIN {X 0,Y 559.914,Z 1167.276,A -85,B 0,C 180,E1 26545.698,E2 26545.698} C_VEL
LIN {X 0,Y 559.914,Z 1163.46,A -85,B 0,C 180,E1 26543.334,E2 26543.334} C_VEL
LIN {X 0,Y 559.955,Z 1158.55,A -85,B 0,C 180,E1 26541.166,E2 26541.166} C_VEL
LIN {X 0,Y 560,Z 1151.763,A -85,B 0,C 180,E1 26538.882,E2 26538.882} C_VEL
LIN {X 0,Y 560.097,Z 1144.108,A -85,B 0,C 180,E1 26536.791,E2 26536.791} C_VEL
LIN {X 0,Y 560.275,Z 1133.881,A -85,B 0,C 180,E1 26534.473,E2 26534.473} C_VEL
LIN {X 0,Y 560.534,Z 1122.818,A -85,B 0,C 180,E1 26532.347,E2 26532.347} C_VEL
LIN {X 0,Y 560.864,Z 1109.751,A -85,B 0,C 180,E1 26530.201,E2 26530.201} C_VEL
LIN {X 0,Y 561.292,Z 1095.341,A -85,B 0,C 180,E1 26528.137,E2 26528.137} C_VEL
LIN {X 0,Y 561.795,Z 1079.939,A -85,B 0,C 180,E1 26526.227,E2 26526.227} C_VEL
LIN {X 0,Y 562.438,Z 1062.112,A -85,B 0,C 180,E1 26524.293,E2 26524.293} C_VEL
LIN {X 0,Y 563.12,Z 1044.254,A -85,B 0,C 180,E1 26522.595,E2 26522.595} C_VEL
LIN {X 0,Y 563.844,Z 1025.334,A -85,B 0,C 180,E1 26521.045,E2 26521.045} C_VEL
LIN {X 0,Y 564.609,Z 1004.598,A -85,B 0,C 180,E1 26519.57,E2 26519.57} C_VEL
LIN {X 0,Y 565.355,Z 984.825,A -85,B 0,C 180,E1 26518.373,E2 26518.373} C_VEL
LIN {X 0,Y 566.072,Z 962.174,A -85,B 0,C 180,E1 26517.22,E2 26517.22} C_VEL
LIN {X 0,Y 566.732,Z 941.497,A -85,B 0,C 180,E1 26516.359,E2 26516.359} C_VEL
LIN {X 0,Y 567.277,Z 918.333,A -85,B 0,C 180,E1 26515.6,E2 26515.6} C_VEL
LIN {X 0,Y 567.748,Z 896.115,A -85,B 0,C 180,E1 26515.058,E2 26515.058} C_VEL
LIN {X 0,Y 568.087,Z 858.62,A -85,B 0,C 180,E1 26514.463,E2 26514.463} C_VEL
LIN {X 0,Y 569.51,Z 652.546,A -85,B 0,C 180,E1 26511.376,E2 26511.376} C_VEL
LIN {X 0,Y 570.046,Z 552.724,A -85,B 0,C 180,E1 26509.825,E2 26509.825} C_VEL
LIN {X 0,Y 567.946,Z 542.47,A -85,B 0,C 180,E1 26509.453,E2 26509.453} C_VEL
LIN {X 0,Y 568.221,Z 531.13,A -85,B 0,C 180,E1 26508.632,E2 26508.632} C_VEL
LIN {X 0,Y 561.928,Z 517.288,A -85,B 0,C 180,E1 26506.996,E2 26506.996} C_VEL
LIN {X 0,Y 560.321,Z 513.868,A -85,B 0,C 180,E1 26506.574,E2 26506.574} C_VEL
LIN {X 0,Y 560.224,Z 513.255,A -85,B 0,C 180,E1 26506.49,E2 26506.49} C_VEL
LIN {X 0,Y 560.249,Z 513.256,A -85,B 0,C 180,E1 26503.119,E2 26503.119} C_VEL
LIN {X 0,Y 560.247,Z 513.263,A -85,B 0,C 180,E1 26499.977,E2 26499.977} C_VEL
LIN {X 0,Y 560.24,Z 513.258,A -85,B 0,C 180,E1 26496.571,E2 26496.571} C_VEL
LIN {X 0,Y 560.278,Z 513.251,A -85,B 0,C 180,E1 26493.343,E2 26493.343} C_VEL
LIN {X 0,Y 560.238,Z 513.253,A -85,B 0,C 180,E1 26490.05,E2 26490.05} C_VEL
LIN {X 0,Y 560.278,Z 513.256,A -85,B 0,C 180,E1 26486.837,E2 26486.837} C_VEL
LIN {X 0,Y 560.247,Z 513.245,A -85,B 0,C 180,E1 26483.563,E2 26483.563} C_VEL
LIN {X 0,Y 560.279,Z 513.251,A -85,B 0,C 180,E1 26480.255,E2 26480.255} C_VEL
LIN {X 0,Y 560.269,Z 513.245,A -85,B 0,C 180,E1 26476.911,E2 26476.911} C_VEL
LIN {X 0,Y 560.268,Z 513.252,A -85,B 0,C 180,E1 26473.52,E2 26473.52} C_VEL
LIN {X 0,Y 560.269,Z 513.249,A -85,B 0,C 180,E1 26470.176,E2 26470.176} C_VEL
LIN {X 0,Y 560.264,Z 513.256,A -85,B 0,C 180,E1 26466.867,E2 26466.867} C_VEL
LIN {X 0,Y 560.264,Z 513.254,A -85,B 0,C 180,E1 26463.581,E2 26463.581} C_VEL
LIN {X 0,Y 560.279,Z 513.259,A -85,B 0,C 180,E1 26460.204,E2 26460.204} C_VEL
LIN {X 0,Y 560.279,Z 513.252,A -85,B 0,C 180,E1 26456.726,E2 26456.726} C_VEL
LIN {X 0,Y 560.255,Z 513.258,A -85,B 0,C 180,E1 26453.441,E2 26453.441} C_VEL
LIN {X 0,Y 560.274,Z 513.249,A -85,B 0,C 180,E1 26450.135,E2 26450.135} C_VEL
LIN {X 0,Y 560.245,Z 513.256,A -85,B 0,C 180,E1 26446.9,E2 26446.9} C_VEL
LIN {X 0,Y 560.278,Z 513.25,A -85,B 0,C 180,E1 26443.622,E2 26443.622} C_VEL
LIN {X 0,Y 560.242,Z 513.254,A -85,B 0,C 180,E1 26440.396,E2 26440.396} C_VEL
LIN {X 0,Y 560.259,Z 513.246,A -85,B 0,C 180,E1 26436.993,E2 26436.993} C_VEL
